// TwinCAT 3 PLC project P637_teljes
// ProgramVersion: 3.1.4023.0
// libraries:
//   Tc2_MC2, * (Beckhoff Automation GmbH)
//   Tc2_NC, * (Beckhoff Automation GmbH)
//   Tc2_SerialCom, * (Beckhoff Automation GmbH)
//   Tc2_Standard, * (Beckhoff Automation GmbH)
//   Tc2_System, * (Beckhoff Automation GmbH)
//   Tc2_TcpIp, * (Beckhoff Automation GmbH)
//   Tc2_Utilities, * (Beckhoff Automation GmbH)
//   Tc3_Module, * (Beckhoff Automation GmbH)
//   VisuDialogs, * (System)
//   Recipe Management,3.5.13.0,System
// project tree:
//   / CheckDivDInt.TcPOU, CheckDivLInt.TcPOU, CheckDivLReal.TcPOU, CheckDivReal.TcPOU, CheckLRangeSigned.TcPOU, CheckLRangeUnsigned.TcPOU, CheckPointer.TcPOU, CheckRangeSigned.TcPOU, CheckRangeUnsigned.TcPOU, GlobalTextList.TcGTLO, ImagePool.TcIPO (not stored), Jozsitengely_task.TcTTO, NTC_Task.TcTTO, Pistitengely_task.TcTTO, PlcTask.TcTTO, RecipeManager.TcRMO (not stored), Robot_task.TcTTO, Visualization Manager.TcVMO (not stored), VISU_TASK.TcTTO
//   DUTs/ ST_RobotState.TcDUT, STATES.TcDUT, User.TcDUT
//   GVLs/ GVL.TcGVL
//   POUs/ AUTOMATA.TcPOU, AUTOMATA_lepesek1.TcTLO, AUTOMATA_lepesek2.TcTLO, CheckBounds.TcPOU, DUT_types.TcTLO, ErrorList.TcTLO, ErrorList1.TcTLO, ErrorList2.TcTLO, JozsiProcess.TcPOU, MAIN.TcPOU
//   POUs/GENERAL/Components/ BARCODE_SCANNER.TcPOU, HEGESZTOK.TcPOU, INIT.TcPOU, RobotProcess.TcPOU, TERMEKVALTAS.TcPOU
//   POUs/GENERAL/Components/Robot/ ROBOTCOMMAND_OLD.TcPOU, ROBOTCOMMAND.TcPOU, ROBOTREMOTE_OLD.TcPOU, ROBOTREMOTE.TcPOU
//   POUs/GENERAL/Helpers/ fb_RobotStatusToBools.TcPOU, fb_SplitRobotResult.TcPOU, f_RobotCommandTranslation.TcPOU, f_RobotNTCTengelytolTavol.TcPOU, f_RobotPtTengelytolTavol.TcPOU, GetResourceFromCommand.TcPOU, f_GetRobotState.TcPOU
//   POUs/GENERAL/Executors/ f_E_Robot.TcPOU
//   POUs/JOZSI/Components/ HAJLITOK.TcPOU, HEGESZTESUTMERES.TcPOU, HEGESZTESUTMERES_1.TcPOU, HEGESZTOFEJTISZTITAS.TcPOU, JOZSITENGELY.TcPOU, KAMERA.TcPOU, NTC.TcPOU, NTCProcess.TcPOU
//   POUs/JOZSI/Executors/ f_E_Tengely.TcPOU
//   POUs/PISTI/Components/ KameraProcess.TcPOU, KAMERAREMOTE.TcPOU, KAPPE.TcPOU, HIMBA.TcPOU, Laser.TcPOU, Laser_old.TcPOU, LOGGING.TcPOU, PISTITENGELY.TcPOU, TEST_R_INTERPOL.TcPOU, ZEBRASCANNER.TcPOU, VEGMERO.TcPOU
//   POUs/PISTI/Helpers/ fb_GetPT1000MinMaxResFromTemp.TcPOU, f_GetNTCMinR.TcPOU, f_GetNTCMaxR.TcPOU, f_GetNTCNomR.TcPOU, f_GetPtMinR.TcPOU, f_GetPtMaxR.TcPOU, f_GetPtNomR.TcPOU, f_GetPtTfromR.TcPOU, f_GetPTTEMPFromRES.TcPOU, f_GetISOLvalue.TcPOU, f_GetNTCMaxTempFromRes.TcPOU, f_GetNTCNomTempFromRes.TcPOU, f_GetNTCMinTempFromRes.TcPOU, REAL_TO_STRING2.TcPOU
//   VISUs/ AddDelete.TcVIS, Biztos.TcVIS, Hegesztes_Karbantartas.TcVIS, Hegesztofej_IOk.TcVIS, Hegesztofej_IOk_Pt.TcVIS, Hegesztofej_IOk_NTC.TcVIS, Himba.TcVIS, Kamera_Pt.TcVIS, Login.TcVIS, Pt1000_oldali_kamera.TcVIS, Hegeszto_statusz.TcVIS, Lezer.TcVIS, Kamera.TcVIS, Robot.TcVIS, Kappe_pres.TcVIS, Start_ablak.TcVIS, Behelyezes.TcVIS, Rendszerinditas.TcVIS, Start_ellenorzes.TcVIS, Tengely_NTC_beallitasok.TcVIS, Tengely_Pt1000.TcVIS, Tengelyek.TcVIS, Tengely_NTC.TcVIS, Tengely_Pt1000_beallitasok.TcVIS, Termektipus.TcVIS, Vegmero.TcVIS, Hegesztes_Tengely_Pt1000.TcVIS, Hegesztes_Tengely_NTC.TcVIS, Kodolvaso.TcVIS, Hajlitok.TcVIS, Szerviz.TcVIS, NTC_szerviz.TcVIS, Hegesztok.TcVIS, Termeles0.TcVIS, Meresek.TcVIS, Beallitasok.TcVIS, Vegmero_idoallando.TcVIS, Vegmero_sokk.TcVIS, Vegmero_teljes.TcVIS, Vegmero_szigeteles.TcVIS, Vegmero_auto.TcVIS, Vegmero_ellenallas.TcVIS, Vegmero_kezi.TcVIS, Visualization_new.TcVIS
// real-time tasks:
//   TASK PlcTask: cycle T#10ms, priority 12, ADS port 350
//   TASK 637Visual: cycle T#20ms, priority 16, ADS port 351
//   TASK Pistitengely_task: cycle T#10ms, priority 13, ADS port 352
//   TASK Jozsitengely_task: cycle T#10ms, priority 14, ADS port 353
//   TASK Robot_task: cycle T#10ms, priority 20, ADS port 354
//   TASK NTC_Task: cycle T#1ms, priority 11, ADS port 355
//   TASK zebra: cycle T#1ms, priority 26, ADS port 356
// motion (NC):
//   TASK NC-Task 1 SAF: cycle T#2ms, priority 4, ADS port 501
//   TASK NC-Task 1 SVB: cycle T#2ms, priority 6, ADS port 511
//   AXIS JozsiTengely (id 1)
//     Dynamic: AccelerationMaximum=25000, DecelerationMaximum=25000, Acceleration=11382.8, Deceleration=11382.8, Jerk=114403
//     Velo: RefSearch=100, RefSync=5, SlowManual=57.2, FastManual=343.2, Fast=1144, Maximum=1144
//     OtherSettings: AllowMotionCmdToSlave=true, PulseDistancePos=200, PulseDistanceNeg=200
//     encoder EncType=19
//       EncPara: ScaleFactorNumerator=20, ScaleFactorDenominator=1048576, MaxCount=#xffffffff
//         Inc: RefMode=1
//     drive DrvType=16
//       DrvPara: MaxCount=#xffffffff, DriveControlDWord=#x00000100
//         Analog: VeloReferenz=1258.4
//         TimeComp: TaskDelayCycles=1
//     controller CtrType=1
//       CtrPara: PriorControlFactor=1
//         PosDiffControl: Enable=false, Range=200
//         Observer: BandWidth=20
//   AXIS PistiTengely (id 2)
//     Dynamic: Acceleration=11325.5840016781, Deceleration=11325.5840016781, Jerk=114411.676767905
//     Velo: RefSearch=100, RefSync=5, SlowManual=57.2, FastManual=343.2, Fast=1144, Maximum=1144
//     OtherSettings: AllowMotionCmdToSlave=true
//     encoder EncType=19
//       EncPara: ScaleFactorNumerator=20, ScaleFactorDenominator=1048576, MaxCount=#xffffffff
//         Inc: RefMode=1
//     drive DrvType=16
//       DrvPara: MaxCount=#xffffffff, DriveControlDWord=#x00000100
//         Analog: VeloReferenz=1200
//         TimeComp: TaskDelayCycles=1
//     controller CtrType=1
//       CtrPara: PriorControlFactor=1
//         PosDiffControl: Enable=false
//         Observer: BandWidth=20
// I/O:
//   DEVICE Device 1 (EtherCAT), AmsNetId 10.0.0.31.2.1
//     Term 1 (EK1200) [EK1200-5000 EtherCAT Power supply (2A E-Bus)]
//       PistiTengely (EL7211-0010) [EL7211-0010 1Ch. MDP742 Servo motor output stage with OCT (50V, 4.5A RMS)]
//       JózsiTengely (EL7211-0010) [EL7211-0010 1Ch. MDP742 Servo motor output stage with OCT (50V, 4.5A RMS)]
//       Útmérők 4 (EL5032) [EL5032 2Ch. EnDat Encoder]
//       Bemenetek (EL1809) [EL1809 16Ch. Dig. Input 24V, 3ms]
//       Bemenetek2 (EL1809) [EL1809 16Ch. Dig. Input 24V, 3ms]
//       Kimenetek (EL2809) [EL2809 16Ch. Dig. Output 24V, 0.5A]
//       Kimenetek2 (EL2809) [EL2809 16Ch. Dig. Output 24V, 0.5A]
//       Hőszenzor (EL3201-0010) [EL3201-0010 1K. Ana. Eingang PT100 (RTD), hochgenau]
//       EtherCatTerminal (EK1122) [EK1122 2 port EtherCAT junction]
//         Pisti Inputs1 (EP1008-0001) [EP1008-0001 8 Ch. Dig. Input 24V, 3ms, M8]
//         Pisti Inputs2 (EP1809-0021) [EP1809-0021 16 Ch. Dig. Input 24V, 3ms, M8]
//         IOLink Box (EP6224-3022) [EP6224-3022 (IO Link Master Class B)]
//         Jozsi Inputs1 (EP1809-0021) [EP1809-0021 16 Ch. Dig. Input 24V, 3ms, M8]
//         Jozsi Inputs2 (EP1809-0021) [EP1809-0021 16 Ch. Dig. Input 24V, 3ms, M8]
//         Végméro (EK1100) [EK1100 EtherCAT Coupler (2A E-Bus)]
//           AnalogIn (EL3068) [EL3068 8Ch. Ana. Input 0-10V]
//           DigitalIn (EL1808) [EL1808 8Ch. Dig. Input 24V, 3ms]
//           DigitalOut (EL2808) [EL2808 8Ch. Dig. Output 24V, 0.5A]
//           Term 18 (EL9011) [EL9011 End Terminal]
// variable links:
//   NC-Task 1 SAF/Axes/JozsiTengely <-> Device 1 (EtherCAT)/Term 1 (EK1200)/JózsiTengely (EL7211-0010)
//     Drive/Inputs/In/nDataIn1 <-> DRV Following error actual value/Following error actual value
//     Drive/Inputs/In/nDcOutputTime <-> InfoData/DcOutputShift
//     Drive/Inputs/In/nState1 <-> DRV Statusword/JozsiStatusword
//     Drive/Inputs/In/nState2 <-> DRV Statusword/JozsiStatusword @bit 8
//     Drive/Inputs/In/nState4 @bit 1 <-> WcState/InputToggle
//     Drive/Inputs/In/nState4 <-> WcState/WcState
//     Drive/Outputs/Out/nCtrl1 <-> DRV Controlword/Controlword
//     Drive/Outputs/Out/nCtrl2 <-> DRV Controlword/Controlword @bit 8
//     Drive/Outputs/Out/nDataOut1 <-> DRV Target position/Target position
//     Enc/Inputs/In/nDataIn1 <-> FB Position/Position
//     Enc/Inputs/In/nDcInputTime <-> InfoData/DcInputShift
//     Enc/Inputs/In/nState4 @bit 1 <-> WcState/InputToggle
//     Enc/Inputs/In/nState4 <-> WcState/WcState
//   NC-Task 1 SAF/Axes/PistiTengely <-> Device 1 (EtherCAT)/Term 1 (EK1200)/PistiTengely (EL7211-0010)
//     Drive/Inputs/In/nDataIn1 <-> DRV Following error actual value/Following error actual value
//     Drive/Inputs/In/nDcOutputTime <-> InfoData/DcOutputShift
//     Drive/Inputs/In/nState1 <-> DRV Statusword/PistiStatusword
//     Drive/Inputs/In/nState2 <-> DRV Statusword/PistiStatusword @bit 8
//     Drive/Inputs/In/nState4 @bit 1 <-> WcState/InputToggle
//     Drive/Inputs/In/nState4 <-> WcState/WcState
//     Drive/Outputs/Out/nCtrl1 <-> DRV Controlword/Controlword
//     Drive/Outputs/Out/nCtrl2 <-> DRV Controlword/Controlword @bit 8
//     Drive/Outputs/Out/nDataOut1 <-> DRV Target position/Target position
//     Enc/Inputs/In/nDataIn1 <-> FB Position/Position
//     Enc/Inputs/In/nDcInputTime <-> InfoData/DcInputShift
//     Enc/Inputs/In/nState4 @bit 1 <-> WcState/InputToggle
//     Enc/Inputs/In/nState4 <-> WcState/WcState
//   P637_teljes/P637_teljes Instance <-> Device 1 (EtherCAT)/Term 1 (EK1200)/Bemenetek (EL1809)
//     NTC_Task Inputs/GVL.bFenysorompoPt <-> Channel 15/FénysorompóPt
//     NTC_Task Inputs/HEGESZTOK.bHegesztoStromFehler <-> Channel 7/HegesztoStromFehler
//     NTC_Task Inputs/MAIN.bLevegoOK <-> Channel 3/LevegoOK
//     NTC_Task Inputs/NTC.bAlarm <-> Channel 12/NTC_Alarm
//     NTC_Task Inputs/NTC.bReady <-> Channel 13/NTC_Ready
//     PlcTask Inputs/GVL.bFenysorompoNTC <-> Channel 16/FénysorompóNTC
//     PlcTask Inputs/GVL.bHeatingTempOK <-> Channel 2/FűtőtőmbHőmOK
//     PlcTask Inputs/HEGESZTOK.bHegesztoBereit <-> Channel 6/HegesztoBereit
//     PlcTask Inputs/HEGESZTOK.bHegesztoFK <-> Channel 14/HegesztoFolyamatKesz
//     PlcTask Inputs/HEGESZTOK.bHegesztoMitStromIn <-> Channel 8/HegesztoMitStrom
//     PlcTask Inputs/VEGMERO.bFedelNyitva <-> Channel 1/VegmeroFedelLecsukásÉrzékelő
//     Robot_task Inputs/HEGESZTOK.bHegesztoElektrodenAnfordem <-> Channel 5/HegesztoElektrodenAnfordem
//     Robot_task Inputs/HEGESZTOK.bHegesztoNichtBereit <-> Channel 9/HegesztoNichtBereit
//     Robot_task Inputs/HEGESZTOK.bHegesztoVorwarnung <-> Channel 4/HegesztoVorwarnung
//     Robot_task Inputs/NTC.bSpeedReached <-> Channel 11/NTC_SpeedReached
//     Robot_task Inputs/NTC.bZeroSpeed <-> Channel 10/NTC_ZeroSpeed
//   P637_teljes/P637_teljes Instance <-> Device 1 (EtherCAT)/Term 1 (EK1200)/Bemenetek2 (EL1809)
//     PlcTask Inputs/GVL.bBiztonsagiFold <-> Channel 5/BiztonságiFöld
//     PlcTask Inputs/GVL.bBiztonsagiTap <-> Channel 6/BiztonságiTáp
//     PlcTask Inputs/GVL.bHegesztoHiba <-> Channel 7/HegesztoHiba
//     PlcTask Inputs/GVL.bKameraHulsePozOK <-> Channel 2/KameraHulsePoz
//     PlcTask Inputs/GVL.bKameraHulseVanOK <-> Channel 1/KameraHulseVan
//     PlcTask Inputs/GVL.bKameraSzinekOK <-> Channel 3/KameraSzinekOK
//     PlcTask Inputs/GVL.bKameraVezetekPozOK <-> Channel 4/KameraTavOK
//     PlcTask Inputs/HIMBA.bHimba_szenzor <-> Channel 10/Himba_szenzor
//     Robot_task Inputs/GVL.bPtKameraHegesztesOK <-> Channel 9/PtKameraHegesztesOK
//   P637_teljes/P637_teljes Instance <-> Device 1 (EtherCAT)/Term 1 (EK1200)/EtherCatTerminal (EK1122)/IOLink Box (EP6224-3022)
//     NTC_Task Outputs/HEGESZTOK.bHegeszto3 <-> IO-Link Port1/Hegeszto
//     NTC_Task Outputs/HEGESZTOK.bHegesztoFejekOutput[0] <-> IO-Link Port3/Hegesztofej1LE
//     NTC_Task Outputs/HEGESZTOK.bHegesztoFejekOutput[1] <-> IO-Link Port3/Hegesztofej2LE
//     NTC_Task Outputs/HEGESZTOK.bHegesztoFejekOutput[2] <-> IO-Link Port3/Hegesztofej3LE
//     NTC_Task Outputs/HEGESZTOK.bHegesztoFejekOutput[3] <-> IO-Link Port3/Valve 4 solenoid 14
//     PlcTask Outputs/GVL.bAdapterLefogo <-> IO-Link Port1/AdapterLefogó
//     PlcTask Outputs/HAJLITOK.bElohajlitoAlso <-> IO-Link Port4/AlsoElohajlito
//     PlcTask Outputs/HAJLITOK.bElohajlitoFelso <-> IO-Link Port4/FelsoElohajlito
//     PlcTask Outputs/HAJLITOK.bVeghajlitoAlso <-> IO-Link Port4/AlsoVeghajlito
//     PlcTask Outputs/HAJLITOK.bVeghajlitoFelso <-> IO-Link Port4/FelsoVeghajlito
//     PlcTask Outputs/HIMBA.bHimba <-> IO-Link Port1/Himba
//     PlcTask Outputs/KAPPE.bKappeBalFelLe <-> IO-Link Port1/KappeprésBal
//     PlcTask Outputs/KAPPE.bKappeFelLe <-> IO-Link Port1/Kappeprés
//     PlcTask Outputs/KAPPE.bKappeJobbFelLe <-> IO-Link Port1/KappeprésJobb
//     PlcTask Outputs/MAIN.bZoliSzelep <-> IO-Link Port4/Valve 5 solenoid 14
//     PlcTask Outputs/NTCProcess.bKiszedo <-> IO-Link Port2/NTC_Kiszedo
//     PlcTask Outputs/NTCProcess.bMegfogo <-> IO-Link Port2/NTC_Megfogo
//     PlcTask Outputs/NTCProcess.bVagoHajlito <-> IO-Link Port2/NTC_VagoHajlito
//     PlcTask Outputs/VEGMERO.bHutesOn <-> IO-Link Port1/HutesBe
//     PlcTask Outputs/VEGMERO.bLezertakaro <-> IO-Link Port1/LézerTakaró
//     PlcTask Outputs/VEGMERO.bMerotukBeKi <-> IO-Link Port1/Mérofej
//     PlcTask Outputs/VEGMERO.bPlatniBalraJobbra <-> IO-Link Port1/PlatniForgat
//     PlcTask Outputs/VEGMERO.bPlatniFelLe <-> IO-Link Port1/PlatniLeFel
//     Robot_task Outputs/GVL.bTempJozsiSzeleptombNTC[{3..7}] <-> IO-Link Port2/Valve {4..8} solenoid 14  (5 links)
//     Robot_task Outputs/GVL.bTempJozsiSzeleptomb[5] <-> IO-Link Port4/Valve 6 solenoid 14
//     Robot_task Outputs/GVL.bTempJozsiSzeleptomb[6] <-> IO-Link Port4/Valve 7 solenoid 14
//     Robot_task Outputs/GVL.bTempJozsiSzeleptomb[7] <-> IO-Link Port4/Valve 8 solenoid 14
//   P637_teljes/P637_teljes Instance <-> Device 1 (EtherCAT)/Term 1 (EK1200)/EtherCatTerminal (EK1122)/Jozsi Inputs1 (EP1809-0021)
//     Jozsitengely_task Inputs/GVL.bJozsiNegSwitch <-> Channel 7/LimitSwitchNeg
//     NTC_Task Inputs/NTC.bNTCLaberzekeloJobb <-> Channel 16/NTCJobbPozicioban
//     NTC_Task Inputs/NTC.bPirosGomb <-> Channel 13/NTCPirosGomb
//     NTC_Task Inputs/NTC.bZoldGomb <-> Channel 14/NTCZöldGomb
//     PlcTask Inputs/GVL.bHegeszto2FentBent <-> Channel 4/Hegeszto2FentBent
//     PlcTask Inputs/GVL.bHegeszto2FentKint <-> Channel 3/Hegeszto2FentKint
//     PlcTask Inputs/GVL.bHegeszto2LentBent <-> Channel 5/Hegeszto2LentBent
//     PlcTask Inputs/GVL.bHegeszto2LentKint <-> Channel 6/Hegeszto2LentKint
//     PlcTask Inputs/JOZSITENGELY.bNTC_OK <-> Channel 15/NTC_OK
//     PlcTask Inputs/NTCProcess.bKiszedoBent <-> Channel 12/NTC_KiszedoBent
//     PlcTask Inputs/NTCProcess.bKiszedoKint <-> Channel 11/NTC_KiszedoKint
//     PlcTask Inputs/NTCProcess.bMegfogoNyitva <-> Channel 9/NTC_MegfogoNyitva
//     PlcTask Inputs/NTCProcess.bMegfogoZarva <-> Channel 10/NTC_MegfogoZarva
//     PlcTask Inputs/NTCProcess.bVagoHajlitoFent <-> Channel 2/NTCVagoFent
//     PlcTask Inputs/NTCProcess.bVagoHajlitoLent <-> Channel 1/NTCVagoLent
//     Robot_task Inputs/GVL.bLimitSwitchNeg <-> Channel 7/LimitSwitchNeg
//     Robot_task Inputs/GVL.bNTCPirosGomb <-> Channel 13/NTCPirosGomb
//     Robot_task Inputs/GVL.bNTCPozicioban <-> Channel 8/NTCBalPozicioban
//     Robot_task Inputs/GVL.bNTCVagoFent <-> Channel 2/NTCVagoFent
//     Robot_task Inputs/GVL.bNTCVagoLent <-> Channel 1/NTCVagoLent
//     Robot_task Inputs/GVL.bNTCZoldGomb <-> Channel 14/NTCZöldGomb
//     Robot_task Inputs/GVL.bNTC_KiszedoBent <-> Channel 12/NTC_KiszedoBent
//     Robot_task Inputs/GVL.bNTC_KiszedoKint <-> Channel 11/NTC_KiszedoKint
//     Robot_task Inputs/GVL.bNTC_MegfogoNyitva <-> Channel 9/NTC_MegfogoNyitva
//     Robot_task Inputs/GVL.bNTC_MegfogoZarva <-> Channel 10/NTC_MegfogoZarva
//     Robot_task Inputs/GVL.bNTC_OK <-> Channel 15/NTC_OK
//     Robot_task Inputs/NTC.bNTCLaberzekeloBal <-> Channel 8/NTCBalPozicioban
//   P637_teljes/P637_teljes Instance <-> Device 1 (EtherCAT)/Term 1 (EK1200)/EtherCatTerminal (EK1122)/Jozsi Inputs2 (EP1809-0021)
//     Jozsitengely_task Inputs/GVL.bJozsiPosSwitch <-> Channel 16/LimitSwitchPlus
//     Jozsitengely_task Inputs/JOZSITENGELY.bJozsiHomeSwitch <-> Channel 16/LimitSwitchPlus
//     PlcTask Inputs/GVL.bHegeszto1BalFent <-> Channel 5/Hegeszto1BalFent
//     PlcTask Inputs/GVL.bHegeszto1BalLent <-> Channel 6/Hegeszto1BalLent
//     PlcTask Inputs/GVL.bHegeszto1JobbFent <-> Channel 13/Hegeszto1JobbFent
//     PlcTask Inputs/GVL.bHegeszto1JobbLent <-> Channel 14/Hegeszto1JobbLent
//     PlcTask Inputs/GVL.bNTCAdapterErzekelo <-> Channel 15/AdapterÉrzékelő
//     PlcTask Inputs/GVL.bPres1AlsoLent <-> Channel 3/Pres1AlsoLent
//     PlcTask Inputs/GVL.bPres2AlsoLent <-> Channel 12/Pres2AlsoLent
//     PlcTask Inputs/GVL.bPres1FelsoFent <-> Channel 2/Pres1FelsoFent
//     PlcTask Inputs/GVL.bPres2FelsoFent <-> Channel 10/Pres2FelsoFent
//     PlcTask Inputs/GVL.bStartNTC <-> Channel 8/StartNTC
//     PlcTask Inputs/HAJLITOK.bElohajlitoAlsoFent <-> Channel 4/Pres1AlsoFent
//     PlcTask Inputs/HAJLITOK.bElohajlitoAlsoLent <-> Channel 3/Pres1AlsoLent
//     PlcTask Inputs/HAJLITOK.bElohajlitoFelsoFent <-> Channel 2/Pres1FelsoFent
//     PlcTask Inputs/HAJLITOK.bElohajlitoFelsoLent <-> Channel 1/Pres1FelsoLent
//     PlcTask Inputs/HAJLITOK.bVeghajlitoAlsoFent <-> Channel 11/Pres2AlsoFent
//     PlcTask Inputs/HAJLITOK.bVeghajlitoAlsoLent <-> Channel 12/Pres2AlsoLent
//     PlcTask Inputs/HAJLITOK.bVeghajlitoFelsoFent <-> Channel 10/Pres2FelsoFent
//     PlcTask Inputs/HAJLITOK.bVeghajlitoFelsoLent <-> Channel 9/Pres2FelsoLent
//     PlcTask Inputs/MAIN.bZoliGomb <-> Channel 7/Input
//     Robot_task Inputs/GVL.bLimitSwitchPlus <-> Channel 16/LimitSwitchPlus
//     Robot_task Inputs/GVL.bPres1AlsoFent <-> Channel 4/Pres1AlsoFent
//     Robot_task Inputs/GVL.bPres2AlsoFent <-> Channel 11/Pres2AlsoFent
//     Robot_task Inputs/GVL.bPres1FelsoLent <-> Channel 1/Pres1FelsoLent
//     Robot_task Inputs/GVL.bPres2FelsoLent <-> Channel 9/Pres2FelsoLent
//   P637_teljes/P637_teljes Instance <-> Device 1 (EtherCAT)/Term 1 (EK1200)/EtherCatTerminal (EK1122)/Pisti Inputs1 (EP1008-0001)
//     NTC_Task Inputs/GVL.bHegeszto3Lent <-> Channel 5/HegesztőLent
//     Pistitengely_task Inputs/GVL.bPistiPosSwitch <-> Channel 6/LimitSwichPlus
//     Pistitengely_task Inputs/PISTITENGELY.bPistiHomeSwitch <-> Channel 6/LimitSwichPlus
//     PlcTask Inputs/GVL.bAdapterLefogoBent <-> Channel 1/AdapterLefogóBent
//     PlcTask Inputs/GVL.bAdapterLefogoKint <-> Channel 2/AdapterLefogóKint
//     PlcTask Inputs/GVL.bAdaptererzekelo <-> Channel 3/Adapterérzékelő
//     PlcTask Inputs/GVL.bHegeszto3Fent <-> Channel 4/HegesztőFent
//     PlcTask Inputs/HIMBA.bHimba_elol <-> Channel 8/Himba_elol
//     PlcTask Inputs/HIMBA.bHimba_hatul <-> Channel 7/Himba_hatul
//     Robot_task Inputs/GVL.bLimitSwichPlus <-> Channel 6/LimitSwichPlus
//     Robot_task Inputs/GVL.bTempPistiInputs1[0] <-> Channel 1/AdapterLefogóBent
//     Robot_task Inputs/GVL.bTempPistiInputs1[1] <-> Channel 2/AdapterLefogóKint
//     Robot_task Inputs/GVL.bTempPistiInputs1[2] <-> Channel 3/Adapterérzékelő
//     Robot_task Inputs/GVL.bTempPistiInputs1[3] <-> Channel 4/HegesztőFent
//     Robot_task Inputs/GVL.bTempPistiInputs1[4] <-> Channel 5/HegesztőLent
//     Robot_task Inputs/GVL.bTempPistiInputs1[5] <-> Channel 6/LimitSwichPlus
//   P637_teljes/P637_teljes Instance <-> Device 1 (EtherCAT)/Term 1 (EK1200)/EtherCatTerminal (EK1122)/Pisti Inputs2 (EP1809-0021)
//     Pistitengely_task Inputs/GVL.bPistiNegSwitch <-> Channel 8/LimitSwitchMinus
//     PlcTask Inputs/GVL.bKappePresFent <-> Channel 15/KappePrésFent
//     PlcTask Inputs/GVL.bKappepresNincsLegalul <-> Channel 7/KappeprésNincsLegalul
//     PlcTask Inputs/KAPPE.bKappeBalFent <-> Channel 11/KappeBalBent
//     PlcTask Inputs/KAPPE.bKappeBalLent <-> Channel 12/KappeBalKint
//     PlcTask Inputs/KAPPE.bKappeJobbFent <-> Channel 10/KappeJobbBent
//     PlcTask Inputs/KAPPE.bKappeJobbLent <-> Channel 9/KappeJobbKint
//     PlcTask Inputs/VEGMERO.bLezertakaroNyitva <-> Channel 6/LézerNyitva
//     PlcTask Inputs/VEGMERO.bLezertakaroZarva <-> Channel 5/LézerZárva
//     PlcTask Inputs/VEGMERO.bMerotukBent <-> Channel 4/MérőBent
//     PlcTask Inputs/VEGMERO.bMerotukKint <-> Channel 3/MérőKint
//     PlcTask Inputs/VEGMERO.bNagyFeszMerotuLent <-> Channel 16/NagyFeszMérőtűLent
//     PlcTask Inputs/VEGMERO.bPlatniBalon <-> Channel 14/PlatniBalon
//     PlcTask Inputs/VEGMERO.bPlatniFent <-> Channel 1/PlatniFent
//     PlcTask Inputs/VEGMERO.bPlatniJobbon <-> Channel 13/PlatniJobbon
//     PlcTask Inputs/VEGMERO.bPlatniLent <-> Channel 2/PlatniLent
//     Robot_task Inputs/GVL.bKappeBalBent <-> Channel 11/KappeBalBent
//     Robot_task Inputs/GVL.bKappeBalKint <-> Channel 12/KappeBalKint
//     Robot_task Inputs/GVL.bKappeJobbBent <-> Channel 10/KappeJobbBent
//     Robot_task Inputs/GVL.bKappeJobbKint <-> Channel 9/KappeJobbKint
//     Robot_task Inputs/GVL.bLezerNyitva <-> Channel 6/LézerNyitva
//     Robot_task Inputs/GVL.bLezerZarva <-> Channel 5/LézerZárva
//     Robot_task Inputs/GVL.bLimitSwitchMinus <-> Channel 8/LimitSwitchMinus
//     Robot_task Inputs/GVL.bMeroBent <-> Channel 4/MérőBent
//     Robot_task Inputs/GVL.bMeroKint <-> Channel 3/MérőKint
//     Robot_task Inputs/GVL.bPlatniBalon <-> Channel 14/PlatniBalon
//     Robot_task Inputs/GVL.bPlatniFent <-> Channel 1/PlatniFent
//     Robot_task Inputs/GVL.bPlatniJobbon <-> Channel 13/PlatniJobbon
//     Robot_task Inputs/GVL.bPlatniLent <-> Channel 2/PlatniLent
//     Robot_task Inputs/KAPPE.bKappeFent <-> Channel 15/KappePrésFent
//     Robot_task Inputs/KAPPE.bKappeNincsLegalul <-> Channel 7/KappeprésNincsLegalul
//   P637_teljes/P637_teljes Instance <-> Device 1 (EtherCAT)/Term 1 (EK1200)/EtherCatTerminal (EK1122)/Végméro (EK1100)/AnalogIn (EL3068)
//     PlcTask Inputs/VEGMERO.NTRES <-> AI Standard Channel 6/NTRES
//     PlcTask Inputs/VEGMERO.NTRES2 <-> AI Standard Channel 8/NTRES2
//     PlcTask Inputs/VEGMERO.PTRES <-> AI Standard Channel 5/PTRES
//     PlcTask Inputs/VEGMERO.U12V <-> AI Standard Channel 1/U12V
//     PlcTask Inputs/VEGMERO.U48V <-> AI Standard Channel 7/U48V
//     PlcTask Inputs/VEGMERO.U600V <-> AI Standard Channel 3/U600V
//     PlcTask Inputs/VEGMERO.U600VExt <-> AI Standard Channel 2/U600VEXT
//     PlcTask Inputs/VEGMERO.UISOL <-> AI Standard Channel 4/UISOL
//   P637_teljes/P637_teljes Instance <-> Device 1 (EtherCAT)/Term 1 (EK1200)/EtherCatTerminal (EK1122)/Végméro (EK1100)/DigitalOut (EL2808)
//     PlcTask Outputs/VEGMERO.PT_SOKK48V <-> Channel 3/PT-SOKK
//     PlcTask Outputs/VEGMERO.b600VBe <-> Channel 1/600VBe
//     PlcTask Outputs/VEGMERO.bRL_ISOL <-> Channel 2/RL-ISOL
//     Robot_task Outputs/GVL.bVentillatorok1Be <-> Channel 7/Ventillatorok1
//     Robot_task Outputs/GVL.bVentillatorok2Be <-> Channel 8/Ventillatorok2
//   P637_teljes/P637_teljes Instance <-> Device 1 (EtherCAT)/Term 1 (EK1200)/Hőszenzor (EL3201-0010)
//     PlcTask Inputs/VEGMERO.iHorzekelo <-> RTD/Value
//   P637_teljes/P637_teljes Instance <-> Device 1 (EtherCAT)/Term 1 (EK1200)/JózsiTengely (EL7211-0010)
//     Jozsitengely_task Inputs/JOZSITENGELY.nAxisStatus <-> DRV Statusword/JozsiStatusword
//   P637_teljes/P637_teljes Instance <-> Device 1 (EtherCAT)/Term 1 (EK1200)/Kimenetek (EL2809)
//     NTC_Task Outputs/HEGESZTOK.bHegesztoMitStromOut <-> Channel 15/HegesztoMitStrom
//     NTC_Task Outputs/HEGESZTOK.bHegesztoProgramValasztoOutput[0] <-> Channel 12/HegesztoPRG0
//     NTC_Task Outputs/HEGESZTOK.bHegesztoProgramValasztoOutput[1] <-> Channel 13/HegesztoPRG1
//     NTC_Task Outputs/HEGESZTOK.bHegesztoProgramValasztoOutput[2] <-> Channel 14/HegesztoPRG2
//     NTC_Task Outputs/HEGESZTOK.bHegesztoProgramValasztoOutput[3] <-> Channel 16/HegesztoPRG3
//     NTC_Task Outputs/HEGESZTOK.bHegesztoStart <-> Channel 10/HegesztoSTART
//     NTC_Task Outputs/HEGESZTOK.bHegesztoValtoOutput[0] <-> Channel 6/HegesztoValto1
//     NTC_Task Outputs/HEGESZTOK.bHegesztoValtoOutput[1] <-> Channel 7/HegesztoValto2
//     NTC_Task Outputs/HEGESZTOK.bHegesztoValtoOutput[2] <-> Channel 8/HegesztoValto3
//     PlcTask Outputs/GVL.bHegesztoHibaTorles <-> Channel 11/HegesztoMeldung
//     PlcTask Outputs/MAIN.bLevego <-> Channel 9/Levego
//     Robot_task Outputs/GVL.bTempOutputs[{0..4}] <-> Channel {1..5}/Output  (5 links)
//   P637_teljes/P637_teljes Instance <-> Device 1 (EtherCAT)/Term 1 (EK1200)/Kimenetek2 (EL2809)
//     NTC_Task Outputs/HEGESZTOK.bHegesztoProgramValasztoOutput[4] <-> Channel 8/HegesztoPRG4
//     NTC_Task Outputs/NTC.bForwardRotationStart <-> Channel 2/NTC_ForwardRotationStart
//     NTC_Task Outputs/NTC.bReverseRotationStart <-> Channel 3/NTC_ReverseRotationStart
//     NTC_Task Outputs/NTC.bServoON <-> Channel 1/NTC_ServoON
//     PlcTask Outputs/GVL.bBiztonsagiZarBe <-> Channel 7/BiztonságiZár
//     PlcTask Outputs/GVL.bElszivasBe <-> Channel 4/bElszivasBe
//     PlcTask Outputs/GVL.bKameraPROG <-> Channel 10/KameraPROG
//     PlcTask Outputs/GVL.bKameraTrigger <-> Channel 9/KameraTrigger
//     PlcTask Outputs/GVL.bPtKameraTrigger <-> Channel 13/PtKameraTrigger
//     Robot_task Outputs/NTC.bNTCFekBal <-> Channel 11/NTCLeftBreak
//     Robot_task Outputs/NTC.bNTCFekJobb <-> Channel 12/NTCRightBreak
//     Robot_task Outputs/NTC.bReset <-> Channel 6/NTC_Reset
//     Robot_task Outputs/NTC.bSpeed1 <-> Channel 5/NTC_Speed1
//   P637_teljes/P637_teljes Instance <-> Device 1 (EtherCAT)/Term 1 (EK1200)/PistiTengely (EL7211-0010)
//     Pistitengely_task Inputs/PISTITENGELY.nAxisStatus <-> DRV Statusword/PistiStatusword
//   P637_teljes/P637_teljes Instance <-> Device 1 (EtherCAT)/Term 1 (EK1200)/Útmérők 4 (EL5032)
//     NTC_Task Inputs/HEGESZTOK.ulHegeszto1Utmero <-> FB Inputs Channel 1/Hegeszto1 Position
//     NTC_Task Inputs/HEGESZTOK.ulHegeszto2Utmero <-> FB Inputs Channel 2/Hegeszto2 Position
//   P637_teljes/P637_teljes Instance <-> NC-Task 1 SAF/Axes/JozsiTengely
//     Jozsitengely_task Inputs/GVL.axisJozsiTengely.NcToPlc <-> Outputs/ToPlc
//     Jozsitengely_task Inputs/JOZSITENGELY.bOperational <-> Outputs/ToPlc/StateDWord/Operational
//     Jozsitengely_task Inputs/JOZSITENGELY.lrJozsiActPos <-> Outputs/ToPlc/ActPos
//     Jozsitengely_task Outputs/GVL.axisJozsiTengely.PlcToNc <-> Inputs/FromPlc
//     Robot_task Inputs/JOZSITENGELY.nJozsiErrorCode <-> Outputs/ToPlc/ErrorCode
//   P637_teljes/P637_teljes Instance <-> NC-Task 1 SAF/Axes/PistiTengely
//     Pistitengely_task Inputs/GVL.axisPistiTengely.NcToPlc <-> Outputs/ToPlc
//     Pistitengely_task Inputs/PISTITENGELY.bOperational <-> Outputs/ToPlc/StateDWord/Operational
//     Pistitengely_task Inputs/PISTITENGELY.lrPistiActPos <-> Outputs/ToPlc/ActPos
//     Pistitengely_task Outputs/GVL.axisPistiTengely.PlcToNc <-> Inputs/FromPlc
//     Robot_task Inputs/PISTITENGELY.nPistiErrorCode <-> Outputs/ToPlc/ErrorCode

CONFIGURATION P637_teljes
    RESOURCE PLC ON TwinCAT3
        TASK Jozsitengely_task(INTERVAL := T#10ms, PRIORITY := 14);
        TASK NTC_Task(INTERVAL := T#1ms, PRIORITY := 11);
        TASK Pistitengely_task(INTERVAL := T#10ms, PRIORITY := 13);
        TASK PlcTask(INTERVAL := T#10ms, PRIORITY := 12);
        TASK Robot_task(INTERVAL := T#10ms, PRIORITY := 20);
        TASK VISU_TASK(INTERVAL := T#20ms, PRIORITY := 16);
        PROGRAM JOZSITENGELY WITH Jozsitengely_task : JOZSITENGELY;
        PROGRAM NTC WITH NTC_Task : NTC;
        PROGRAM HEGESZTESUTMERES WITH NTC_Task : HEGESZTESUTMERES;
        PROGRAM ZEBRASCANNER WITH NTC_Task : ZEBRASCANNER;
        PROGRAM HEGESZTOK WITH NTC_Task : HEGESZTOK;
        PROGRAM PISTITENGELY WITH Pistitengely_task : PISTITENGELY;
        PROGRAM MAIN WITH PlcTask : MAIN;
        PROGRAM Laser WITH PlcTask : Laser;
        PROGRAM VEGMERO WITH PlcTask : VEGMERO;
        PROGRAM HAJLITOK WITH PlcTask : HAJLITOK;
        PROGRAM NTCProcess WITH PlcTask : NTCProcess;
        PROGRAM KAPPE WITH PlcTask : KAPPE;
        PROGRAM AUTOMATA WITH PlcTask : AUTOMATA;
        PROGRAM HEGESZTOFEJTISZTITAS WITH PlcTask : HEGESZTOFEJTISZTITAS;
        PROGRAM INIT WITH PlcTask : INIT;
        PROGRAM LOGGING WITH PlcTask : LOGGING;
        PROGRAM TERMEKVALTAS WITH PlcTask : TERMEKVALTAS;
        PROGRAM KAMERA WITH PlcTask : KAMERA;
        PROGRAM HIMBA WITH PlcTask : HIMBA;
        PROGRAM KameraProcess WITH PlcTask : KameraProcess;
        PROGRAM KAMERAREMOTE WITH PlcTask : KAMERAREMOTE;
        PROGRAM BARCODE_SCANNER WITH PlcTask : BARCODE_SCANNER;
        PROGRAM RobotProcess WITH Robot_task : RobotProcess;
        PROGRAM ROBOTREMOTE WITH Robot_task : ROBOTREMOTE;
        PROGRAM ROBOTCOMMAND WITH Robot_task : ROBOTCOMMAND;
        PROGRAM VisuElems_Visu_Prg WITH VISU_TASK : VisuElems.Visu_Prg;
    END_RESOURCE
END_CONFIGURATION

// ---- DUTs/ST_RobotState.TcDUT
TYPE ST_RobotState :
STRUCT
	sResult: STRING;
	bVakuumSzippantoFent: BOOL;
	bVakuumSzippantoLent: BOOL;
	bCsipeszNyitva: BOOL;
	bCsipeszZarva: BOOL;
	bVakuumA: BOOL;
	bVakuumB: BOOL;
	rX: REAL;
	rY: REAL;
	rZ: REAL;
	rU: REAL;
	sHand: STRING;
END_STRUCT
END_TYPE

// ---- DUTs/STATES.TcDUT
{attribute 'qualified_only'}
{attribute 'strict'}
TYPE STATES :
(
	enum_member := 0
);
END_TYPE

// ---- DUTs/User.TcDUT
TYPE User:
	STRUCT
		UserID: INT;
		UserNumber: STRING;
		UserName: STRING;
		UserLevel: INT;
		UserExist: BOOL;
	END_STRUCT
END_TYPE

// ---- GVLs/GVL.TcGVL
{attribute 'qualified_only'}
VAR_GLOBAL
	
	//Felhasználók beállítása
	AddDelButtonDis: BOOL;
	LogButtonsDis: BOOL;
	Logout_Button: BOOL;
	AddDeleteEnabled: BOOL;
	LoginEnabled: BOOL;
	
	UserID_Elozo: INT;
	UserID_Temp: INT;
	UserTemp: User;
	UserActual: User;
	UserNotFound: BOOL;
	UserModify: BOOL;
	UserDelete: BOOL;

	Biztos: BOOL;
	
	//Persistent data változói
	bStart_WrPer: BOOL;
	bError_WrPer: BOOL;
	fbWritePersistentData: WritePersistentData;
	bBusy_WrPer: BOOL;
	
	//System
	EngineExecuteList : ARRAY[1..5] OF STRING;
	bSettingsAutoSaveElozo: BOOL;
	bSettingsAutoSave: BOOL;
	
	//Temp
//	bTempInputs AT %I*: ARRAY [0..15] OF BOOL;
	bHeatingTempOK AT %I*: BOOL;
	bTempOutputs AT %Q*: ARRAY [0..15] OF BOOL;
	
	// Kamera I/O-k
	bKameraTrigger AT %Q*: BOOL;
	bKameraPROG AT %Q*: BOOL;
	bKameraBusy AT %I*: BOOL;
	bKameraHulseVanOK AT %I*: BOOL;
	bKameraHulsePozOK AT %I*: BOOL;
	bKameraSzinekOK AT %I*: BOOL;
	bKameraVezetekPozOK AT %I*: BOOL;
	bPtKameraTrigger AT %Q*: BOOL;
	bPtKameraHegesztesOK AT %I*: BOOL;
	
	// Hegesztő I/O-k
	bHegesztoHiba AT %I*: BOOL;
	bHegesztoHibaTorles AT %Q*: BOOL;

	// Hegesztési beállítás
	nWeldingDeformation1: DINT;
	nWeldingDeformation2: DINT;
	nWeldingDeformation3: DINT;
	nWeldingDeformation4: DINT;
	nWeldingDeformation5: DINT;
	bAutomaticWeldingStop1Elozo: BOOL;
	bAutomaticWeldingStop1: BOOL;
	bAutomaticWeldingStop2Elozo: BOOL;
	bAutomaticWeldingStop2: BOOL;
	bAutomaticWeldingStop3Elozo: BOOL;
	bAutomaticWeldingStop3: BOOL;
	bAutomaticWeldingStop4Elozo: BOOL;
	bAutomaticWeldingStop4: BOOL;
	bAutomaticWeldingStop5Elozo: BOOL;
	bAutomaticWeldingStop5: BOOL;
	nWeldingStopDistance1Elozo: DINT := 320;
	nWeldingStopDistance1: DINT := 320;
	nWeldingDistanceMin1Elozo: DINT := 320;
	nWeldingDistanceMin1: DINT := 320;
	nWeldingDistanceMax1Elozo: DINT := 320;
	nWeldingDistanceMax1: DINT := 320;
	nWeldingStopDistance2Elozo: DINT := 320;
	nWeldingStopDistance2: DINT := 320;
	nWeldingDistanceMin2Elozo: DINT := 320;
	nWeldingDistanceMin2: DINT := 320;
	nWeldingDistanceMax2Elozo: DINT := 320;
	nWeldingDistanceMax2: DINT := 320;
	nWeldingStopDistance3Elozo: DINT := 320;
	nWeldingStopDistance3: DINT := 320;
	nWeldingDistanceMin3Elozo: DINT := 320;
	nWeldingDistanceMin3: DINT := 320;
	nWeldingDistanceMax3Elozo: DINT := 320;
	nWeldingDistanceMax3: DINT := 320;
	nWeldingStopDistance4Elozo: DINT := 320;
	nWeldingStopDistance4: DINT := 320;
	nWeldingDistanceMin4Elozo: DINT := 320;
	nWeldingDistanceMin4: DINT := 320;
	nWeldingDistanceMax4Elozo: DINT := 320;
	nWeldingDistanceMax4: DINT := 320;
	nWeldingStopDistance5Elozo: DINT := 320;
	nWeldingStopDistance5: DINT := 320;
	nWeldingDistanceMin5Elozo: DINT := 320;
	nWeldingDistanceMin5: DINT := 320;
	nWeldingDistanceMax5Elozo: DINT := 320;
	nWeldingDistanceMax5: DINT := 320;
	nWeldingStopDistance1_637: DINT := 320;
	nWeldingDistanceMin1_637: DINT := 320;
	nWeldingDistanceMax1_637: DINT := 320;
	nWeldingStopDistance2_637: DINT := 320;
	nWeldingDistanceMin2_637: DINT := 320;
	nWeldingDistanceMax2_637: DINT := 320;
	nWeldingStopDistance3_637: DINT := 320;
	nWeldingDistanceMin3_637: DINT := 320;
	nWeldingDistanceMax3_637: DINT := 320;
	nWeldingStopDistance4_637: DINT := 320;
	nWeldingDistanceMin4_637: DINT := 320;
	nWeldingDistanceMax4_637: DINT := 320;
	nWeldingStopDistance5_637: DINT := 320;
	nWeldingDistanceMin5_637: DINT := 320;
	nWeldingDistanceMax5_637: DINT := 320;
	nWeldingStopDistance1_745: DINT := 320;
	nWeldingDistanceMin1_745: DINT := 320;
	nWeldingDistanceMax1_745: DINT := 320;
	nWeldingStopDistance2_745: DINT := 320;
	nWeldingDistanceMin2_745: DINT := 320;
	nWeldingDistanceMax2_745: DINT := 320;
	nWeldingStopDistance3_745: DINT := 320;
	nWeldingDistanceMin3_745: DINT := 320;
	nWeldingDistanceMax3_745: DINT := 320;
	nWeldingStopDistance4_745: DINT := 320;
	nWeldingDistanceMin4_745: DINT := 320;
	nWeldingDistanceMax4_745: DINT := 320;
	nWeldingStopDistance5_745: DINT := 320;
	nWeldingDistanceMin5_745: DINT := 320;
	nWeldingDistanceMax5_745: DINT := 320;
	ulWeldingStartDistance1: ULINT;
	ulWeldingStartDistance2: ULINT;
	ulWeldingStartDistance3: ULINT;
	ulWeldingStartDistance4: ULINT;
	ulWeldingStartDistance5: ULINT;
	nWeldingDistanceStartMin1Elozo: DINT := 0;
	nWeldingDistanceStartMin1: DINT := 0;
	nWeldingDistanceStartMax1Elozo: DINT := 210000;
	nWeldingDistanceStartMax1: DINT := 210000;
	nWeldingDistanceStartMin2Elozo: DINT := 0;
	nWeldingDistanceStartMin2: DINT := 0;
	nWeldingDistanceStartMax2Elozo: DINT := 210000;
	nWeldingDistanceStartMax2: DINT := 210000;
	nWeldingDistanceStartMin3Elozo: DINT := 0;
	nWeldingDistanceStartMin3: DINT := 0;
	nWeldingDistanceStartMax3Elozo: DINT := 210000;
	nWeldingDistanceStartMax3: DINT := 210000;
	nWeldingDistanceStartMin4Elozo: DINT := 0;
	nWeldingDistanceStartMin4: DINT := 0;
	nWeldingDistanceStartMax4Elozo: DINT := 210000;
	nWeldingDistanceStartMax4: DINT := 210000;
	nWeldingDistanceStartMin5Elozo: DINT := 0;
	nWeldingDistanceStartMin5: DINT := 0;
	nWeldingDistanceStartMax5Elozo: DINT := 210000;
	nWeldingDistanceStartMax5: DINT := 210000;
	bWeldingLog: BOOL;
	bWeldingLogElozo: BOOL;
	nElectrode1UsageElozo: DINT;
	nElectrode1Usage: DINT;
	nElectrode1UsageMaxElozo: DINT := 1;
	nElectrode1UsageMax: DINT := 1;
	nElectrode1UsageWarnElozo: DINT := 1;
	nElectrode1UsageWarn: DINT := 1;
	nElectrode1AlarmColor: DWORD := 16#FFFFFF00;
	nElectrode2UsageElozo: DINT;
	nElectrode2Usage: DINT;
	nElectrode2UsageMaxElozo: DINT := 1;
	nElectrode2UsageMax: DINT := 1;
	nElectrode2UsageWarnElozo: DINT := 1;
	nElectrode2UsageWarn: DINT := 1;
	nElectrode2AlarmColor: DWORD := 16#FF8F8F00;
	nElectrode3UsageElozo: DINT;
	nElectrode3Usage: DINT;
	nElectrode3UsageMaxElozo: DINT := 1;
	nElectrode3UsageMax: DINT := 1;
	nElectrode3UsageWarnElozo: DINT := 1;
	nElectrode3UsageWarn: DINT := 1;
	nElectrode3AlarmColor: DWORD := 16#FF8F8F00;
	
	nHegFejTisztCiklusokElozo: UINT := 5;
	nHegFejTisztCiklusok: UINT := 5;
	nHegFejTisztProgramElozo: UINT := 11;
	nHegFejTisztProgram: UINT := 11;
	
	//Pisti Globals
	axisPistiTengely: AXIS_REF;
	bPistiPosSwitch AT %I*: BOOL;
	bPistiNegSwitch AT %I*: BOOL;
	bPistiServo : BOOL := TRUE;
	bTempPistiInputs1 AT %I*: ARRAY [0..7] OF BOOL;
	bHimbaOK: BOOL := FALSE;
	bAdapterLefogoBent AT %I*: BOOL; // 0
	bAdapterLefogoKint AT %I*: BOOL; // 1
	bAdaptererzekelo AT %I*: BOOL; // 2
	bHegeszto3Fent AT %I*: BOOL; // 3
	bHegeszto3Lent AT %I*: BOOL; // 4
	bLimitSwichPlus AT %I*: BOOL; // 5
	bStartPt AT %I*: BOOL; // 6
	bInput_7: BOOL; // 7 
//	bTempPistiInputs2 AT %I*: ARRAY [0..15] OF BOOL;
	bPlatniFent AT %I*: BOOL; // 0
	bPlatniLent AT %I*: BOOL; // 1
	bMeroKint AT %I*: BOOL; // 2
	bMeroBent AT %I*: BOOL; // 3
	bLezerZarva AT %I*: BOOL; // 4
	bLezerNyitva AT %I*: BOOL; // 5
	bKappepresNincsLegalul AT %I*: BOOL; // 6
	bLimitSwitchMinus AT %I*: BOOL; // 7
	bKappeJobbKint AT %I*: BOOL; // 8
	bKappeJobbBent AT %I*: BOOL; // 9
	bKappeBalBent AT %I*: BOOL; // 10
	bKappeBalKint AT %I*: BOOL; // 11
	bPlatniJobbon AT %I*: BOOL; // 12
	bPlatniBalon AT %I*: BOOL; // 13
	bKappePresFent AT %I*: BOOL; // 14
	bInput_15: BOOL; // 15
//	bTempPistiOutputs1 AT %Q*: ARRAY [0..9] OF BOOL;
	bAdapterLefogo AT %Q*: BOOL; // 0
	bJOZSITENGELYReserved: BOOL;
	lrPtSzervizboxElozo : LREAL := -5;
	lrPtSzervizbox : LREAL := -5;
	lrNTCSzervizboxElozo : LREAL := -10;
	lrNTCSzervizbox : LREAL := -10;
	lrHajlitoPosition1Elozo : LREAL := -401.2;
	lrHajlitoPosition1 : LREAL := -401.2;
	lrHajlitoPosition2Elozo : LREAL := -575.1;
	lrHajlitoPosition2 : LREAL := -575.1;
	lrHegesztoPosition1Elozo : LREAL := -789.0;
	lrHegesztoPosition1 : LREAL := -789.0;
	lrHegesztoPosition2Elozo : LREAL := -792.0;
	lrHegesztoPosition2 : LREAL := -792.0;
	lrHegesztoPosition3Elozo : LREAL := -794.7;
	lrHegesztoPosition3 : LREAL := -794.7;
	lrCsiszoloPosition1Elozo : LREAL := -780;
	lrCsiszoloPosition1 : LREAL := -780;
	lrCsiszoloPosition2Elozo : LREAL := -800;
	lrCsiszoloPosition2 : LREAL := -800;
	lrHegesztoPosition4Elozo : LREAL := -1109.913;
	lrHegesztoPosition4 : LREAL := -1109.913;
	lrHegesztoPosition5Elozo : LREAL := -1101.15;
	lrHegesztoPosition5 : LREAL := -1101.15;
	lrHegesztoPosition6Elozo : LREAL := -379.7;
	lrHegesztoPosition6 : LREAL := -379.7;
	lrHegesztoPosition7Elozo : LREAL := -386;
	lrHegesztoPosition7 : LREAL := -386;
	lrNTCKameraPositionElozo : LREAL := -160.622;
	lrNTCKameraPosition : LREAL := -160.622;
	lrPtKameraPositionElozo : LREAL := -503.4;
	lrPtKameraPosition : LREAL := -503.4;
	lrRobotKappePositionElozo : LREAL := -694.5;
	lrRobotKappePosition : LREAL := --694.5;
	lrKodolvasasPositionElozo: LREAL := -841.54;
	lrKodolvasasPosition: LREAL := -841.54;
	lrKodolvasasPosition2Elozo: LREAL := -841.54;
	lrKodolvasasPosition2: LREAL := -841.54;
	lrKappePositionElozo : LREAL := -837.11;
	lrKappePosition : LREAL := -837.11;
	lrVegmeroPositionElozo : LREAL := -1054.776;
	lrVegmeroPosition : LREAL := -1054.776;
	
	//Jozsi Globals
	axisJozsiTengely: AXIS_REF;
	bJozsiPosSwitch AT %I*: BOOL;
	bJozsiNegSwitch AT %I*: BOOL;
	bJozsiServo : BOOL := TRUE;
//	bTempJozsiInputs1 AT %I*: ARRAY [0..15] OF BOOL;
	bNTCVagoLent AT %I*: BOOL; // 0
	bNTCVagoFent AT %I*: BOOL; // 1
	bHegeszto2FentKint AT %I*: BOOL; // 2
	bHegeszto2FentBent AT %I*: BOOL; // 3
	bHegeszto2LentBent AT %I*: BOOL; // 4
	bHegeszto2LentKint AT %I*: BOOL; // 5
	bLimitSwitchNeg AT %I*: BOOL; // 6
	bNTCPozicioban AT %I*: BOOL; // 7
	bNTC_MegfogoNyitva AT %I*: BOOL; // 8
	bNTC_MegfogoZarva AT %I*: BOOL; // 9
	bNTC_KiszedoKint AT %I*: BOOL; // 10
	bNTC_KiszedoBent AT %I*: BOOL; // 11
	bNTCPirosGomb AT %I*: BOOL; // 12
	bNTCZoldGomb AT %I*: BOOL; // 13
	bNTC_OK AT %I*: BOOL; // 14
	bNC_15: BOOL; // 15
//	bTempJozsiInputs2 AT %I*: ARRAY [0..15] OF BOOL;
	bPres1FelsoLent AT %I*: BOOL; // 0
	bPres1FelsoFent AT %I*: BOOL; // 1
	bPres1AlsoLent AT %I*: BOOL; // 2
	bPres1AlsoFent AT %I*: BOOL; // 3
	bHegeszto1BalFent AT %I*: BOOL; // 4
	bHegeszto1BalLent AT %I*: BOOL; // 5
	bStartNTC AT %I*: BOOL; // 6
	bInput7: BOOL; // 7
	bPres2FelsoLent AT %I*: BOOL; // 8
	bPres2FelsoFent AT %I*: BOOL; // 9
	bPres2AlsoFent AT %I*: BOOL; // 10
	bPres2AlsoLent AT %I*: BOOL; // 11
	bHegeszto1JobbFent AT %I*: BOOL; // 12
	bHegeszto1JobbLent AT %I*: BOOL; // 13
	bNTCAdapterErzekelo AT %I*: BOOL; // 14
	bLimitSwitchPlus AT %I*: BOOL; // 15
	bTempJozsiSzeleptombNTC AT %Q*: ARRAY [0..7] OF BOOL;
	bTempJozsiSzeleptomb AT %Q*: ARRAY [0..7] OF BOOL;
	bPISTITENGELYReserved: BOOL;
	bHegesztofejTisztitas: BOOL := FALSE;
	
	
	
	//Laser
	bLaserCommOpen : BOOL := FALSE;
	
	//Recipe Manager
	RecipeManagerCommands: RecipeManCommands;
	
	//Mérés
	bEtalonOn : BOOL := TRUE;
	bFedelOK : BOOL :=FALSE;
	bPTResOK : BOOL := FALSE;
	iPTResQ : BYTE :=0;
	bNTCResOK : BOOL := FALSE;
	bNTCRes2OK : BOOL := FALSE;
	iNTCResQ : BYTE := 0;
	iNTC2ResQ : BYTE := 0;
	bIsolOK : BOOL := FALSE;
	iIsolQ : BYTE := 0;
	bTimeConstOK : BOOL := FALSE;
	iTimeConstQ : BYTE := 0;
	bShockOK : BOOL := FALSE;
	iShockQ : BYTE := 0;
	bMarkingOK : BOOL := FALSE;
	bMarking_ellenorizve : BOOL;
	iMarkingQ : BYTE := 0;
	bProduct1OK : BOOL := FALSE;
	bProduct1NOK : BOOL := FALSE;
	bProductOK : BOOL := FALSE;
	bProductNOK : BOOL := FALSE;
	rTemp : REAL := 0;
	rPtRes : REAL := 0;
	rPtResShock : REAL;
	rPtDevElozo : REAL := 2;
	rPtDev : REAL := 2;
	rNTCRes : REAL :=0;
	rNTCRes2 : REAL :=0;
	rNTCDevElozo : REAL := 7;
	rNTCDev : REAL := 7;
	rNTC2DevElozo : REAL := 7;
	rNTC2Dev : REAL := 7;
	rISOL_MAXElozo : REAL := 0.97;
	rISOL_MAX : REAL := 0.97;
	rTempMaxElozo : REAL := 300.0;	// Fűtőtömb hőmérséklete
	rTempMax : REAL := 300.0;	// Fűtőtömb hőmérséklete
	rIdoallandoMaxElozo : REAL :=6;
	rIdoallandoMax : REAL :=6;
	rTimeConst : REAL :=0;
	PTRES_SOKK_MAXElozo : REAL := 2000.0;
	PTRES_SOKK_MAX : REAL := 2000.0;
	iSelectedProductType: INT :=-1;
	iPreviousSelectedProductType: INT :=-1;
	iCurrentProductType: INT :=-3;
	
	//Termelés
	nProductCount1 : DINT;
	nGoodProductCount1 : DINT;
	nBadProductCount1 : DINT;
	nGoodProductCount : DINT;
	nBadProductCount : DINT;
	sProductTypeName : STRING;
	saProductTypeNames: ARRAY[-3..0] OF STRING := ['6379XX_ETALON1', '6379XX_ETALON2',
					 '6379XX_ETALON3','637900'];
	saProductTypeNames745: ARRAY[-3..0] OF STRING := ['7459XX_ETALON1', '7459XX_ETALON2',
					 '7459XX_ETALON3','745900'];
	sNTCType: STRING;
	sPtType: STRING;
	sProductType: STRING;
	sNTCTypeElozo: STRING;
	sPtTypeElozo: STRING;
	sProductTypeElozo: STRING;
	bProductTypeOK: BOOL;

	bElszivasBe AT %Q*: BOOL;
	bSystemStarted: BOOL := FALSE;
	bSystemNotStarted: BOOL := TRUE;

	bHimbaBe: BOOL := FALSE;
	bKameraBe: BOOL := TRUE;
	bHajlitasBe: BOOL := TRUE;
	bHegesztes1Be: BOOL := TRUE;
	bHegesztes2Be: BOOL := TRUE;
	bHegesztes3Be: BOOL := TRUE;
	bHegesztes4Be: BOOL := TRUE;
	bHegesztes5Be: BOOL := TRUE;
	bKameraVegBe: BOOL := TRUE;
	bHegesztes6Be: BOOL := TRUE;
	bHegesztes7Be: BOOL := TRUE;
	bPtKameraBe: BOOL := FALSE;
	bRobotKappeBe: BOOL := TRUE;
	bKappeBe: BOOL := TRUE;
	bMeresBe: BOOL := TRUE;
	bJelolesBe: BOOL := TRUE;
	bNTCInditasFenysorompoval: BOOL;
	bPtInditasFenysorompoval: BOOL;
	sNTCKameraImageID: STRING := 'NTCKamera_NG_Image';
	iBitmap_Version: INT :=0;
	bNTCKameraElfogadva: BOOL := FALSE;
	bNTCKameraNemJo: BOOL := FALSE;
	bNTCEredmenyGombokRejtve: BOOL := TRUE;
	bNTCBezarGombRejtve: BOOL := TRUE;

	// Dátum, időpont
	sYear: STRING;
	sMonth: STRING;
	sDay: STRING;
	sHour: STRING;
	sMinute: STRING;
	sSecond: STRING;
	sDateTime: STRING;
	
	// GUI kezelés
	bMeresiEredmenyekRejtve: BOOL := TRUE;
	bKameraEredmenyekRejtve: BOOL := TRUE;
	bRegiFelulet: BOOL := FALSE;
	iFoLapozo: INT;
	iSzervizLapozo: INT;
	iTengelyLapozo: INT;
	iHegesztoLapozo: INT;
	iMeresLapozo: INT;
	iAutoMeresLapozo: INT;
	
	// Hibakezelés
	bHibauzenetNTCRejtve: BOOL;
	bHibauzenetPtRejtve: BOOL;
	bHibauzenetKozosRejtve: BOOL;
	nHibaKodNTC: UINT;
	nHibaKodPt: UINT;
	nHibaKodKozos: UINT;
	
	// Robot állapot
	stRobotStatusz: ST_RobotState;
	bRobotPaused: BOOL;
	
	// Biztonság
	bFenysorompoNTC AT %I*: BOOL;
	bFenysorompoPt AT %I*: BOOL;
	bBiztonsagiFold AT %I*: BOOL;
	bBiztonsagiTap AT %I*: BOOL;
	bBiztonsagiZarBe AT %Q*: BOOL;
	bVentillatorok1Be AT %Q*: BOOL := TRUE;
	bVentillatorok2Be AT %Q*: BOOL := TRUE;
	
	bBiztonsagiZarGomb: BOOL;
	nHibaKodRobot: UINT;
END_VAR
VAR_GLOBAL CONSTANT
	saProductTypes: ARRAY[-1..16] OF STRING := ['', '637900', '637910', '637920', '637930', '637901', '637911', '637921', '637931','521950','745900','745910','745905','745915','745906','745916','745907','745917'];
	NTC_Sensing_NomRT: ARRAY[0..1, 0..25] OF REAL := 
	[15, 16, 17, 18, 19, 20, 21, 22, 23, 24, 25, 26, 27, 28, 29, 30, 31, 32, 33, 34, 35, 36, 37, 38, 39, 40,
	15660.6, 14955.5, 14286.1, 13650.4, 13046.5, 12472.7, 11927.3, 11408.7, 10915.6, 10446.4, 10000, 9575.1, 9170.5, 8785.3, 8418.3, 8068.6, 7735.3, 7417.5, 7114.5, 6825.5, 6549.8, 6286.7, 6035.5, 5795.6, 5566.6, 5347.8];
	Pt_NomRT: ARRAY[0..1, 0..15] OF REAL := 
	[0,20,40,60,80,100,120,140,160,180,200,220,240,260,280,300,
	1000,1077.9,1155.4,1232.4,1309,1385.1,1460.7,1535.8,1610.5,1684.8,1758.6,1831.9,1904.7,1977.1,2049.1,2120.5];
	
	TERMELES_FUL: INT := 0;
	BEALLITASOK_FUL: INT := 1;
	SZERVIZ_FUL: INT := 2;
	RENDSZERIND_FUL: INT :=0;
	BEHELYEZES_FUL: INT := 1;
	TENGELYEK_FUL: INT := 2;
		NTC_TENGELY_FUL: INT := 0;
		PT_TENGELY_FUL: INT := 1;
	HAJLITOK_FUL: INT := 3;
	HEGESZTES_FUL: INT := 4;
		HEGESZTO_STATUSZ_FUL: INT := 2;
	ROBOT_FUL: INT := 5;
	NTC_VAGO_FUL: INT := 6;
	KAPPE_PRES_FUL: INT := 7;
	VEGMERO_FUL: INT := 8;
	LEZER_FUL: INT := 9;
	KODOLVASO_FUL: INT := 10;
	
	UserLevels: ARRAY[0..3] OF STRING := ['N/A', 'Operátor', 'Csoportvezető', 'Admin'];
	
END_VAR
VAR_GLOBAL PERSISTENT
	Users: ARRAY[0..99] OF User;
END_VAR

// ---- POUs/JOZSI/Components/JOZSITENGELY.TcPOU
PROGRAM JOZSITENGELY
VAR
	JozsiHome: MC_Home;
	bJozsiHomeEnable: BOOL := FALSE;
	bAxisBusy : BOOL := FALSE;
	bAxisActive: BOOL := FALSE;
	bAxisAborted: BOOL := FALSE;
	bAxisError: BOOL := FALSE;
	nAxisErrorID: UDINT;
	bAxisStopDone: BOOL := FALSE;
	bJozsiHomeSwitch AT %I*: BOOL;
	fbJozsiTengelyStop: MC_Stop;
	fbJozsitengelyServo: MC_Power;
	bJozsiPosSwitch : BOOL := TRUE;
	bJozsiTengelySzabad : BOOL;
	bOperational AT %I*: BOOL;
	bNTC_OK AT %I*: BOOL;
	bHomeReady : BOOL := FALSE;
	nAxisStatus AT %I*: UINT;
	bAxisReady : BOOL;
	bAxisOn : BOOL;
	
	//HOME
	bAxisHomeDone: BOOL;
	bAxisHomeBusy: BOOL;
	bAxisHomeActive: BOOL;
	bAxisHomeAborted: BOOL;
	bAxisHomeError: BOOL;
	nAxisHomeErrorID: UDINT;
	
	//MOVE
	bAxisMoveDone: BOOL;
	bAxisMoveBusy: BOOL;
	bAxisMoveActive: BOOL;
	bAxisMoveAborted: BOOL;
	bAxisMoveError: BOOL;
	nAxisMoveErrorID: UDINT;
	
	//COMMAND
	bAxisCommandDone: BOOL;
	bAxisCommandBusy: BOOL;
	bAxisCommandActive: BOOL;
	bAxisCommandAborted: BOOL;
	bAxisCommandError: BOOL;
	nAxisCommandErrorID: UDINT;
	
	
	fbJozsitengelyJOG: MC_Jog;
	bJozsiJOGPlus : BOOL := FALSE;
	bJozsiJOGMinus : BOOL := FALSE;
	fbJozsitengelyReset: MC_Reset;
	bJozsiReset: BOOL;
	nJozsiErrorCode AT %I*: UDINT;
	lrJozsiActPos AT %I*: LREAL;
	fbJozsiMoveAbsolute: MC_MoveAbsolute;
	
	//Pozíciók
//	lrSzervizbox : LREAL := -10;
//	lrHajlitoPosition1 : LREAL := -401.510;
//	lrHajlitoPosition2 : LREAL := -575.44;
//	lrHegesztoPosition1 : LREAL := -789.1;
//	lrHegesztoPosition2 : LREAL := -792.3;
//	lrHegesztoPosition3 : LREAL := -795.1;
//	lrHegesztoPosition4 : LREAL := -1109.913;
//	lrHegesztoPosition5 : LREAL := -1101.15;
//	lrSardisajatPosition1 : LREAL := -756;
//	lrSardisajatPosition2 : LREAL := -738;
	lrSardisajatPosition1 : LREAL := -656;
	lrSardisajatPosition2 : LREAL := -638;
	bJozsiTengelySzabad_TON: TON;
END_VAR
VAR_INPUT
	lrJozsiPosition : LREAL := 0;
	sJozsiAxisCommand: STRING := '';	
END_VAR
VAR_OUTPUT
	n_OutErrId: UINT;
END_VAR

bJozsiTengelySzabad := GVL.bPres1AlsoLent AND GVL.bPres1FelsoFent
						AND GVL.bPres2FelsoFent AND GVL.bPres2AlsoLent
						AND ((GVL.bHegeszto1BalFent AND GVL.bHegeszto1JobbFent) OR GVL.bHegesztofejTisztitas)
						AND GVL.bHegeszto2FentBent AND GVL.bHegeszto2LentBent AND bOperational
//						AND ((GVL.stRobotStatusz.rX>-100) 
//								OR (GVL.stRobotStatusz.rY>350)
//								OR (GVL.stRobotStatusz.rZ>-111))
						AND f_RobotNTCTengelytolTavol()
						AND (GVL.bFenysorompoNTC
							OR (sJozsiAxisCommand='HOME')
							OR (JOZSITENGELY.lrJozsiActPos>-10)
							OR (JOZSITENGELY.lrJozsiActPos<-500))
						AND NOT GVL.bBiztonsagiFold AND GVL.bBiztonsagiTap;
bJozsiTengelySzabad_TON(IN:=bJozsiTengelySzabad, PT:=T#100MS);
IF bJozsiTengelySzabad_TON.Q = FALSE THEN
	IF MAIN.bLevegoOK=FALSE THEN
		n_OutErrId := 5;
	ELSIF GVL.bPres1AlsoLent=FALSE THEN
		n_OutErrId := 149;
	ELSIF GVL.bPres1FelsoFent=FALSE THEN
		n_OutErrId := 147;
	ELSIF GVL.bPres2FelsoFent=FALSE THEN
		n_OutErrId := 163;
	ELSIF GVL.bPres2AlsoLent=FALSE THEN
		n_OutErrId := 167;
	ELSIF GVL.bHegeszto1BalFent=FALSE THEN
		n_OutErrId := 153;
	ELSIF GVL.bHegeszto1JobbFent=FALSE THEN
		n_OutErrId := 169;
	ELSIF GVL.bHegeszto2FentBent=FALSE THEN
		n_OutErrId := 119;
	ELSIF GVL.bHegeszto2LentBent=FALSE THEN
		n_OutErrId := 121;
	ELSIF bOperational=FALSE THEN
		n_OutErrId := 193;
//	ELSIF NOT ((GVL.stRobotStatusz.rX>-100)
//		OR (GVL.stRobotStatusz.rY>350)
//		OR (GVL.stRobotStatusz.rZ>-111)) THEN
	ELSIF NOT f_RobotNTCTengelytolTavol() THEN
		n_OutErrId := 302;
	ELSIF GVL.bFenysorompoNTC=FALSE THEN
		n_OutErrId := 31;
	ELSIF GVL.bBiztonsagiFold=TRUE THEN
		n_OutErrId := 42;
	ELSIF GVL.bBiztonsagiTap=FALSE THEN
		n_OutErrId := 43;
	END_IF
ELSE
	n_OutErrId := 0;
END_IF
bAxisReady:=nAxisStatus MOD 2 = 1;
bAxisOn:=nAxisStatus/2 MOD 2 = 1;

fbJozsiTengelyStop(
	Axis:= GVL.axisJozsiTengely, 
	Execute:= (NOT((GVL.bJozsiPosSwitch OR sJozsiAxisCommand='HOME') AND GVL.bJozsiNegSwitch AND bJozsiTengelySzabad_TON.Q)
				OR (sJozsiAxisCommand='STOP')), 
	Deceleration:= , 
	Jerk:= , 
	Options:= , 
	Done=> bAxisStopDone, 
	Busy=> bAxisBusy, 
	Active=> bAxisActive, 
	CommandAborted=> bAxisAborted, 
	Error=> bAxisError, 
	ErrorID=> nAxisErrorID);
IF (sJozsiAxisCommand='STOP') AND bAxisStopDone AND NOT bAxisError THEN
	sJozsiAxisCommand := '';
END_IF
IF NOT(GVL.bJozsiPosSwitch OR sJozsiAxisCommand='HOME') OR NOT(GVL.bJozsiNegSwitch) THEN
	GVL.bJozsiServo := FALSE;
	sJozsiAxisCommand:='';
END_IF
fbJozsitengelyServo(
	Axis:= GVL.axisJozsiTengely, 
	Enable:= GVL.bJozsiServo, 
	Enable_Positive:= (GVL.bJozsiPosSwitch OR sJozsiAxisCommand='HOME'), 
	Enable_Negative:= GVL.bJozsiNegSwitch, 
	Override:= 100, 
	BufferMode:= , 
	Options:= , 
	Status=> , 
	Busy=> , 
	Active=> , 
	Error=> , 
	ErrorID=> );
	
	//Home
JozsiHome(
	Axis:= GVL.axisJozsiTengely, 
	Execute:= sJozsiAxisCommand='HOME' AND bJozsiTengelySzabad_TON.Q, 
	Position:= DEFAULT_HOME_POSITION, 
	HomingMode:= MC_DefaultHoming, 
	BufferMode:= , 
	Options:= , 
	bCalibrationCam:= NOT(bJozsiHomeSwitch), 
	Done=> bAxisHomeDone, 
	Busy=> bAxisHomeBusy, 
	Active=> bAxisHomeActive, 
	CommandAborted=> bAxisHomeAborted, 
	Error=> bAxisHomeError, 
	ErrorID=> nAxisHomeErrorID);
	//Lefutás ellenőrzése
IF (bAxisHomeDone AND NOT(bAxisHomeBusy OR bAxisHomeActive OR bAxisHomeAborted OR bAxisHomeError)) THEN
	lrJozsiPosition:=GVL.lrNTCSzervizbox;
	sJozsiAxisCommand := 'MOVE';
	bHomeReady:=TRUE;
END_IF
	
	//Move
fbJozsiMoveAbsolute(
	Axis:= GVL.axisJozsiTengely, 
	Execute:= sJozsiAxisCommand='MOVE' AND bJozsiTengelySzabad_TON.Q AND bHomeReady, 
	Position:= lrJozsiPosition, // -1115...0
	Velocity:= 1000, 
	Acceleration:= 0, 
	Deceleration:= 0, 
	Jerk:= 0, 
	BufferMode:= , 
	Options:= , 
	Done=> bAxisMoveDone, 
	Busy=> bAxisMoveBusy, 
	Active=> bAxisMoveActive, 
	CommandAborted=> bAxisMoveAborted, 
	Error=> bAxisMoveError, 
	ErrorID=> nAxisMoveErrorID);
	//Lefutás ellenőrzése
IF (bAxisMoveDone AND NOT(bAxisMoveBusy OR bAxisMoveActive OR bAxisMoveAborted OR bAxisMoveError)) THEN
	sJozsiAxisCommand := '';
END_IF
	
	//JOG
	fbJozsitengelyJOG(
	Axis:= GVL.axisJozsiTengely, 
	JogForward:= bJozsiJOGPlus AND bJozsiTengelySzabad_TON.Q, 
	JogBackwards:= bJozsiJOGMinus AND bJozsiTengelySzabad_TON.Q, 
	Mode:= MC_JOGMODE_STANDARD_SLOW, 
	Position:= , 
	Velocity:= 100, 
	Acceleration:= 0, 
	Deceleration:= 0, 
	Jerk:= 0, 
	Done=> bAxisCommandDone, 
	Busy=> bAxisCommandBusy, 
	Active=> bAxisCommandActive, 
	CommandAborted=> bAxisCommandAborted, 
	Error=> bAxisCommandError, 
	ErrorID=> nAxisCommandErrorID);
	
	//RESET ERROR
	fbJozsitengelyReset(
	Axis:= GVL.axisJozsiTengely, 
	Execute:= bJozsiReset, 
	Done=> bAxisCommandDone, 
	Busy=> bAxisCommandBusy, 
	Error=> bAxisCommandError, 
	ErrorID=> nAxisCommandErrorID);
	
	//Ha nem szabad futtatni
//	IF(NOT(bJozsiTengelySzabad)) THEN
//		sJozsiAxisCommand:='!INTERRUPTED';
//	END_IF

END_PROGRAM

// ---- POUs/GENERAL/Helpers/f_RobotNTCTengelytolTavol.TcPOU
FUNCTION f_RobotNTCTengelytolTavol : BOOL

f_RobotNTCTengelytolTavol:=(GVL.stRobotStatusz.rX>-100) 
							OR (GVL.stRobotStatusz.rY>350)
							OR (GVL.stRobotStatusz.rZ>-111);

END_FUNCTION

// ---- POUs/MAIN.TcPOU
PROGRAM MAIN
VAR_INPUT
	bLevego AT %Q*: BOOL := FALSE;	
END_VAR
VAR_OUTPUT
	bLevegoOK AT %I*: BOOL;	
END_VAR
VAR
	bZoliGomb AT %I* : BOOL;
	bZoliSzelep AT %Q*: BOOL := FALSE;

	bPartsReadReady: BOOL;	
	bSettingsReadReady: BOOL;	
	iInd: INT;
	bTypeFound: BOOL;

	iState: INT:=3;
	sPartsString: STRING;
	sPartsGetStr: T_MaxString;
	iStateS: INT:=3;
	sSettingsString: T_MaxString;
	sSettingsGetStr: T_MaxString;
	iEqu: INT;

	// Fájlnyitás
	bPartsOpenExecute: BOOL := FALSE;
	PartsOpen: fb_FileOpen;
	nPartsOpenMode: DWORD;
	bPartsOpenBusy: BOOL;
	bPartsOpenError: BOOL;
	nPartsOpenError: UDINT;
	hPartsFile: UINT;
	
	bSettingsOpenExecute: BOOL := FALSE;
	SettingsOpen: fb_FileOpen;
	nSettingsOpenMode: DWORD;
	bSettingsOpenBusy: BOOL;
	bSettingsOpenError: BOOL;
	nSettingsOpenError: UDINT;
	hSettingsFile: UINT;
	
	// Fájlírás
	PartsPutStr: fb_FilePuts;
	bPartsPutStrExecute: BOOL;
	bPartsPutStrBusy: BOOL;
	bPartsPutStrError: BOOL;
	nPartsPutStrError: UDINT;
	
	SettingsPutStr: fb_FilePuts;
	bSettingsPutStrExecute: BOOL;
	bSettingsPutStrBusy: BOOL;
	bSettingsPutStrError: BOOL;
	nSettingsPutStrError: UDINT;

	// Fájlolvasás
	PartsGetStr: fb_FileGets;
	bPartsGetStrExecute: BOOL;
	bPartsGetStrBusy: BOOL;
	bPartsGetStrError: BOOL;
	nPartsGetStrError: UDINT;

	SettingsGetStr: fb_FileGets;
	bSettingsGetStrExecute: BOOL;
	bSettingsGetStrBusy: BOOL;
	bSettingsGetStrError: BOOL;
	nSettingsGetStrError: UDINT;
	
	// Fájlzárás
	PartsClose: fb_FileClose;
	bPartsCloseExecute: BOOL;
	bPartsCloseBusy: BOOL;
	bPartsCloseError: BOOL;
	nPartsCloseError: UDINT;

	SettingsClose: fb_FileClose;
	bSettingsCloseExecute: BOOL;
	bSettingsCloseBusy: BOOL;
	bSettingsCloseError: BOOL;
	nSettingsCloseError: UDINT;

	bGetStrPartsEOF: BOOL;
	bGetStrSettingsEOF: BOOL;
	raParameters: ARRAY[0..25] OF REAL;
	Ind: INT;
	sParName: STRING;
	sParValue: STRING;
	sParLine: STRING;
	R_TRIG_BiztZar: R_TRIG;
	
	F_TRIG_BiztZar: F_TRIG;
	TON_Biztzar: TON;
	TON_Biztzar_Start: BOOL;
END_VAR

GVL.fbWritePersistentData(
						NETID:='10.0.0.31.1.1',
						PORT:=851,
						START:=GVL.bStart_WrPer,
						TMOUT:=T#1S,
						BUSY=>GVL.bBusy_WrPer,
						ERR=>GVL.bError_WrPer);


IF (NOT GVL.bBusy_WrPer OR GVL.bError_WrPer) AND GVL.bStart_WrPer THEN
	GVL.bStart_WrPer:=FALSE;
END_IF


IF bZoliGomb=TRUE THEN
	bZoliSzelep := TRUE;
ELSE
	bZoliSzelep := FALSE;
END_IF

TON_Biztzar(IN:=TON_Biztzar_Start, PT:=T#200MS);
R_TRIG_BiztZar(CLK:=GVL.bBiztonsagiZarGomb);
F_TRIG_BiztZar(CLK:=GVL.bBiztonsagiZarGomb);

IF F_TRIG_BiztZar.Q THEN
//	WHILE NOT (ROBOTREMOTE.sRobotCommand='') DO
//		;
//	END_WHILE
//	ROBOTREMOTE.sRobotCommand := 'Pause';
//	ROBOTREMOTE.bRobotCommandSend := TRUE;
	GVL.bBiztonsagiZarBe:=FALSE;
//
END_IF

IF R_TRIG_BiztZar.Q THEN
//	WHILE NOT (ROBOTREMOTE.sRobotCommand='') DO
//		;
//	END_WHILE
	GVL.bBiztonsagiZarBe:=TRUE;
	TON_Biztzar_Start:=TRUE;
//	ROBOTREMOTE.sRobotCommand := 'Continue';
//	ROBOTREMOTE.bRobotCommandSend := TRUE;
END_IF
IF TON_Biztzar.Q THEN
	ROBOTREMOTE.sRobotCommand := 'Continue';
	ROBOTREMOTE.bRobotCommandSend := TRUE;
	TON_Biztzar_Start:=FALSE;
END_IF


CASE iState OF
	2:	// Alkatrészváltozás figyelése
		IF NOT((GVL.sNTCType=GVL.sNTCTypeElozo)
			AND (GVL.sPtType=GVL.sPtTypeElozo)
			AND (GVL.sProductType=GVL.sProductTypeElozo)) THEN
			GVL.bProductTypeOK:=FALSE;	
			IF NOT(GVL.sNTCType=GVL.sNTCTypeElozo) THEN
				IF (LEN(GVL.sNTCType)=32) THEN
					GVL.sNTCType:=RIGHT(GVL.sNTCType,23);
					GVL.sNTCType:=LEFT(GVL.sNTCType,6);
					iState:=3;
				ELSE
					GVL.sNTCType:='HIBÁS KÓD';
				END_IF;
				GVL.sNTCTypeElozo:=GVL.sNTCType;
			END_IF;
			IF NOT(GVL.sPtType=GVL.sPtTypeElozo) THEN
				IF (LEN(GVL.sPtType)=32) THEN
					GVL.sPtType:=RIGHT(GVL.sPtType,23);
					GVL.sPtType:=LEFT(GVL.sPtType,6);
					iState:=3;
				ELSE
					GVL.sPtType:='HIBÁS KÓD';
				END_IF;
				GVL.sPtTypeElozo:=GVL.sPtType;
			END_IF;
			IF NOT(GVL.sProductType=GVL.sProductTypeElozo) THEN
				IF NOT ((GVL.sProductType='637900')
					OR (GVL.sProductType='637901')
					OR (GVL.sProductType='637910')
					OR (GVL.sProductType='637911')
					OR	(GVL.sProductType='637920')
					OR (GVL.sProductType='637921')
					OR (GVL.sProductType='637930')
					OR (GVL.sProductType='637931')
					OR (GVL.sProductType='745900')
					OR (GVL.sProductType='745905')
					OR (GVL.sProductType='745906')
					OR (GVL.sProductType='745907')
					OR (GVL.sProductType='745910')
					OR (GVL.sProductType='745915')
					OR (GVL.sProductType='745916')
					OR (GVL.sProductType='745917')
					OR	(GVL.sProductType='521950')) THEN
					GVL.sProductType:='HIBÁS KÓD';
					GVL.iSelectedProductType:=-1;					
				END_IF
				GVL.sProductTypeElozo:=GVL.sProductType;
			END_IF;
			GVL.bProductTypeOK:=
			(((GVL.sProductType='637900') OR (GVL.sProductType='637901') OR (GVL.sProductType='745900') OR (GVL.sProductType='745910'))
				AND ((GVL.sNTCType='567604') OR (GVL.sNTCType='637707')) AND (GVL.sPtType='637710'))
			OR	(((GVL.sProductType='637910') OR (GVL.sProductType='637911') OR (GVL.sProductType='745905') OR (GVL.sProductType='745915'))
				AND ((GVL.sNTCType='567604') OR (GVL.sNTCType='637707')) AND (GVL.sPtType='637711'))
			OR	(((GVL.sProductType='637920') OR (GVL.sProductType='637921') OR (GVL.sProductType='745907') OR (GVL.sProductType='745917'))
				AND ((GVL.sNTCType='509647') OR (GVL.sNTCType='637700')) AND (GVL.sPtType='637710'))
			OR	(((GVL.sProductType='637930') OR (GVL.sProductType='637931') OR (GVL.sProductType='745906') OR (GVL.sProductType='745916'))
				AND ((GVL.sNTCType='509647') OR (GVL.sNTCType='637700')) AND (GVL.sPtType='637711'))
			OR	(GVL.sProductType='521950');
			IF GVL.bProductTypeOK=TRUE THEN
				bTypeFound:=FALSE;
				iInd:=0;
				WHILE (NOT bTypeFound) AND (iInd<11) DO
					IF GVL.sProductType=GVL.saProductTypes[iInd] THEN
						bTypeFound:=TRUE;
						GVL.iSelectedProductType:=iInd; // Ezzel kezdeményezzük a termékváltást
					ELSE
						iInd:=iInd+1;
					END_IF
				END_WHILE
				IF GVL.iSelectedProductType=8 THEN
					Laser.s_InCommand:='SETJOB_521';
				ELSIF GVL.iSelectedProductType<8 THEN
					Laser.s_InCommand:='SETJOB_637';
					GVL.bKameraPROG:=FALSE;
					GVL.nWeldingStopDistance1:=GVL.nWeldingStopDistance1_637;
					GVL.nWeldingStopDistance2:=GVL.nWeldingStopDistance2_637;
					GVL.nWeldingStopDistance3:=GVL.nWeldingStopDistance3_637;
					GVL.nWeldingStopDistance4:=GVL.nWeldingStopDistance4_637;
					GVL.nWeldingStopDistance5:=GVL.nWeldingStopDistance5_637;
					GVL.nWeldingDistanceMin1:=GVL.nWeldingDistanceMin1_637;
					GVL.nWeldingDistanceMin2:=GVL.nWeldingDistanceMin2_637;
					GVL.nWeldingDistanceMin3:=GVL.nWeldingDistanceMin3_637;
					GVL.nWeldingDistanceMin4:=GVL.nWeldingDistanceMin4_637;
					GVL.nWeldingDistanceMin5:=GVL.nWeldingDistanceMin5_637;
					GVL.nWeldingDistanceMax1:=GVL.nWeldingDistanceMax1_637;
					GVL.nWeldingDistanceMax2:=GVL.nWeldingDistanceMax2_637;
					GVL.nWeldingDistanceMax3:=GVL.nWeldingDistanceMax3_637;
					GVL.nWeldingDistanceMax4:=GVL.nWeldingDistanceMax4_637;
					GVL.nWeldingDistanceMax5:=GVL.nWeldingDistanceMax5_637;
				ELSIF GVL.iSelectedProductType>8 THEN
					GVL.bKameraPROG:=TRUE;
					GVL.nWeldingStopDistance1:=GVL.nWeldingStopDistance1_745;
					GVL.nWeldingStopDistance2:=GVL.nWeldingStopDistance2_745;
					GVL.nWeldingStopDistance3:=GVL.nWeldingStopDistance3_745;
					GVL.nWeldingStopDistance4:=GVL.nWeldingStopDistance4_745;
					GVL.nWeldingStopDistance5:=GVL.nWeldingStopDistance5_745;
					GVL.nWeldingDistanceMin1:=GVL.nWeldingDistanceMin1_745;
					GVL.nWeldingDistanceMin2:=GVL.nWeldingDistanceMin2_745;
					GVL.nWeldingDistanceMin3:=GVL.nWeldingDistanceMin3_745;
					GVL.nWeldingDistanceMin4:=GVL.nWeldingDistanceMin4_745;
					GVL.nWeldingDistanceMin5:=GVL.nWeldingDistanceMin5_745;
					GVL.nWeldingDistanceMax1:=GVL.nWeldingDistanceMax1_745;
					GVL.nWeldingDistanceMax2:=GVL.nWeldingDistanceMax2_745;
					GVL.nWeldingDistanceMax3:=GVL.nWeldingDistanceMax3_745;
					GVL.nWeldingDistanceMax4:=GVL.nWeldingDistanceMax4_745;
					GVL.nWeldingDistanceMax5:=GVL.nWeldingDistanceMax5_745;
					IF GVL.iSelectedProductType>8 AND GVL.iSelectedProductType MOD 2=1 THEN // 74590X
						Laser.s_InCommand:='SETJOB_745900';
					ELSIF GVL.iSelectedProductType>8 AND GVL.iSelectedProductType MOD 2=0 THEN // 74591X
						Laser.s_InCommand:='SETJOB_745910';
					END_IF
				END_IF
			END_IF
		END_IF
	3:	// "Parts" fájl megnyitásának kezdeményezése
		bPartsOpenExecute:=TRUE;
		IF bPartsReadReady=TRUE THEN
			nPartsOpenMode:=FOPEN_MODETEXT OR FOPEN_MODEWRITE;
		ELSE
			nPartsOpenMode:=FOPEN_MODETEXT OR FOPEN_MODEREAD;
		END_IF;
		iState:=4;
	4:	// Várakozás a busy jelre
		IF bPartsOpenBusy=TRUE THEN
			iState:=5;
		END_IF
	5:	// Várakozás a fájlnyitás befejeztére
		IF bPartsOpenBusy=FALSE THEN
			bPartsOpenExecute:=FALSE;
			IF bPartsReadReady=TRUE THEN
				iState:=6;
			ELSE
				iState:=26;
			END_IF
		END_IF
	6:	// Fájlnyitás sikerességének vizsgálata
		IF bPartsOpenError=FALSE THEN
			sPartsString:=CONCAT('NTC=',
							CONCAT(GVL.sNTCType,
							CONCAT('$R$N',
							CONCAT('PT1000=',GVL.sPtType))));
			iState:=7;
		ELSE
			iState:=101;
		END_IF
	7:	// Parts fájlba írás kezdeményezése
		bPartsPutStrExecute:=TRUE;
		iState:=8;
	8:	// Várakozás a busy jelre
		IF bPartsPutStrBusy=TRUE THEN
			iState:=9;
		END_IF
	9:	// Várakozás a fájlírás befejeztére
		IF bPartsPutStrBusy=FALSE THEN
			bPartsPutStrExecute:=FALSE;
			iState:=10;
		END_IF
	10:	// Fájlírás sikerességének vizsgálata
		IF bPartsPutStrError=FALSE THEN
			iState:=11;
		ELSE
			iState:=103;
		END_IF
	26:	// Fájlnyitás sikerességének vizsgálata
		IF bPartsOpenError=FALSE THEN
			iState:=27;
		ELSE
			iState:=101;
		END_IF
	27:	// Parts fájlból olvasás kezdeményezése
		bPartsGetStrExecute:=TRUE;
		iState:=28;
	28:	// Várakozás a busy jelre
		IF bPartsGetStrBusy=TRUE THEN
			iState:=29;
		END_IF
	29:	// Várakozás a fájlolvasás befejeztére
		IF bPartsGetStrBusy=FALSE THEN
			bPartsGetStrExecute:=FALSE;
			iState:=30;
		END_IF
	30:	// Fájlolvasás sikerességének vizsgálata
		IF bPartsGetStrError=FALSE THEN
			IF FIND(sPartsGetStr,'NTC')>0 THEN
				GVL.sNTCType:=LEFT(RIGHT(sPartsGetStr,LEN(sPartsGetStr)-FIND(sPartsGetStr,'=')),6);
				GVL.sNTCTypeElozo:=GVL.sNTCType;
			ELSIF FIND(sPartsGetStr,'PT1000')>0 THEN
				GVL.sPtType:=LEFT(RIGHT(sPartsGetStr,LEN(sPartsGetStr)-FIND(sPartsGetStr,'=')),6);
				GVL.sPtTypeElozo:=GVL.sPtType;
			END_IF
			IF bGetStrPartsEOF=FALSE THEN
				iState:=27;
			ELSE
				iState:=11;
			END_IF
		ELSE
			iState:=103;
		END_IF
	11:	// Parts fájl zárásának kezdeményezése
		bPartsCloseExecute:=TRUE;
		iState:=12;
	12:	// Várakozás a busy jelre
		IF bPartsCloseBusy=TRUE THEN
			iState:=13;
		END_IF
	13:	// Várakozás a fájlzárás befejeztére
		IF bPartsCloseBusy=FALSE THEN
			bPartsCloseExecute:=FALSE;
			iState:=14;
		END_IF
	14:	// Fájlzárás sikerességének vizsgálata
		IF bPartsCloseError=FALSE THEN
			bPartsReadReady:=TRUE;	
			iState:=2;
		ELSE
			iState:=104;
		END_IF
END_CASE

CASE iStateS OF
	2:	// Paraméterváltozás figyelése
		IF (GVL.bSettingsAutoSave=TRUE) AND
			NOT((GVL.bSettingsAutoSave=GVL.bSettingsAutoSaveElozo)
			AND (GVL.rNTCDev=GVL.rNTCDevElozo)
			AND (GVL.rNTC2Dev=GVL.rNTC2DevElozo)
			AND (GVL.rPtDev=GVL.rPtDevElozo)
			AND (GVL.rISOL_MAX=GVL.rISOL_MAXElozo)
			AND (GVL.rTempMax=GVL.rTempMaxElozo)
			AND (GVL.rIdoallandoMax=GVL.rIdoallandoMaxElozo)
			AND (GVL.PTRES_SOKK_MAX=GVL.PTRES_SOKK_MAXElozo)
			AND (GVL.lrPtSzervizbox=GVL.lrPtSzervizboxElozo)
			AND (GVL.lrHegesztoPosition6=GVL.lrHegesztoPosition6Elozo)
			AND (GVL.lrHegesztoPosition7=GVL.lrHegesztoPosition7Elozo)
			AND (GVL.lrRobotKappePosition=GVL.lrRobotKappePositionElozo)
			AND (GVL.lrKappePosition=GVL.lrKappePositionElozo)
			AND (GVL.lrKodolvasasPosition=GVL.lrKodolvasasPositionElozo)
			AND (GVL.lrKodolvasasPosition2=GVL.lrKodolvasasPosition2Elozo)
			AND (GVL.lrVegmeroPosition=GVL.lrVegmeroPositionElozo)
			AND (GVL.lrNTCSzervizbox=GVL.lrNTCSzervizboxElozo)
			AND (GVL.lrHajlitoPosition1=GVL.lrHajlitoPosition1Elozo)
			AND (GVL.lrHajlitoPosition2=GVL.lrHajlitoPosition2Elozo)
			AND (GVL.lrHegesztoPosition1=GVL.lrHegesztoPosition1Elozo)
			AND (GVL.lrHegesztoPosition2=GVL.lrHegesztoPosition2Elozo)
			AND (GVL.lrHegesztoPosition3=GVL.lrHegesztoPosition3Elozo)
			AND (GVL.lrHegesztoPosition4=GVL.lrHegesztoPosition4Elozo)
			AND (GVL.lrHegesztoPosition5=GVL.lrHegesztoPosition5Elozo)
			AND (GVL.nWeldingStopDistance1=GVL.nWeldingStopDistance1Elozo)
			AND (GVL.nWeldingStopDistance2=GVL.nWeldingStopDistance2Elozo)
			AND (GVL.nWeldingStopDistance3=GVL.nWeldingStopDistance3Elozo)
			AND (GVL.nWeldingStopDistance4=GVL.nWeldingStopDistance4Elozo)
			AND (GVL.nWeldingStopDistance5=GVL.nWeldingStopDistance5Elozo)
			AND (GVL.bAutomaticWeldingStop1=GVL.bAutomaticWeldingStop1Elozo)
			AND (GVL.bAutomaticWeldingStop2=GVL.bAutomaticWeldingStop2Elozo)
			AND (GVL.bAutomaticWeldingStop3=GVL.bAutomaticWeldingStop3Elozo)
			AND (GVL.bAutomaticWeldingStop4=GVL.bAutomaticWeldingStop4Elozo)
			AND (GVL.bAutomaticWeldingStop5=GVL.bAutomaticWeldingStop5Elozo)
			AND (GVL.nWeldingDistanceMin1=GVL.nWeldingDistanceMin1Elozo)
			AND (GVL.nWeldingDistanceMin2=GVL.nWeldingDistanceMin2Elozo)
			AND (GVL.nWeldingDistanceMin3=GVL.nWeldingDistanceMin3Elozo)
			AND (GVL.nWeldingDistanceMin4=GVL.nWeldingDistanceMin4Elozo)
			AND (GVL.nWeldingDistanceMin5=GVL.nWeldingDistanceMin5Elozo)
			AND (GVL.nWeldingDistanceMax1=GVL.nWeldingDistanceMax1Elozo)
			AND (GVL.nWeldingDistanceMax2=GVL.nWeldingDistanceMax2Elozo)
			AND (GVL.nWeldingDistanceMax3=GVL.nWeldingDistanceMax3Elozo)
			AND (GVL.nWeldingDistanceMax4=GVL.nWeldingDistanceMax4Elozo)
			AND (GVL.nWeldingDistanceMax5=GVL.nWeldingDistanceMax5Elozo)
			AND (GVL.lrNTCKameraPosition=GVL.lrNTCKameraPositionElozo)
			AND (GVL.lrPtKameraPosition=GVL.lrPtKameraPositionElozo)
			AND (GVL.nWeldingDistanceStartMin1=GVL.nWeldingDistanceStartMin1Elozo)
			AND (GVL.nWeldingDistanceStartMin2=GVL.nWeldingDistanceStartMin2Elozo)
			AND (GVL.nWeldingDistanceStartMin3=GVL.nWeldingDistanceStartMin3Elozo)
			AND (GVL.nWeldingDistanceStartMin4=GVL.nWeldingDistanceStartMin4Elozo)
			AND (GVL.nWeldingDistanceStartMin5=GVL.nWeldingDistanceStartMin5Elozo)
			AND (GVL.nWeldingDistanceStartMax1=GVL.nWeldingDistanceStartMax1Elozo)
			AND (GVL.nWeldingDistanceStartMax2=GVL.nWeldingDistanceStartMax2Elozo)
			AND (GVL.nWeldingDistanceStartMax3=GVL.nWeldingDistanceStartMax3Elozo)
			AND (GVL.nWeldingDistanceStartMax4=GVL.nWeldingDistanceStartMax4Elozo)
			AND (GVL.nWeldingDistanceStartMax5=GVL.nWeldingDistanceStartMax5Elozo)
			AND (GVL.lrCsiszoloPosition1=GVL.lrCsiszoloPosition1Elozo)
			AND (GVL.lrCsiszoloPosition2=GVL.lrCsiszoloPosition2Elozo)
			AND (GVL.nElectrode1Usage=GVL.nElectrode1UsageElozo)
			AND (GVL.nElectrode1UsageMax=GVL.nElectrode1UsageMaxElozo)
			AND (GVL.nElectrode1UsageWarn=GVL.nElectrode1UsageWarnElozo)
			AND (GVL.nElectrode2Usage=GVL.nElectrode2UsageElozo)
			AND (GVL.nElectrode2UsageMax=GVL.nElectrode2UsageMaxElozo)
			AND (GVL.nElectrode2UsageWarn=GVL.nElectrode2UsageWarnElozo)
			AND (GVL.nElectrode3Usage=GVL.nElectrode3UsageElozo)
			AND (GVL.nElectrode3UsageWarn=GVL.nElectrode3UsageWarnElozo)
			AND (GVL.nElectrode3UsageMax=GVL.nElectrode3UsageMaxElozo)
			AND (GVL.nHegFejTisztCiklusok=GVL.nHegFejTisztCiklusokElozo)
			AND (GVL.nHegFejTisztProgram=GVL.nHegFejTisztProgramElozo)
			AND (GVL.bWeldingLog=GVL.bWeldingLogElozo)) THEN
			iStateS:=3;
		END_IF
	3:	// "Parts" fájl megnyitásának kezdeményezése
		bSettingsOpenExecute:=TRUE;
		IF bSettingsReadReady=TRUE THEN
			nSettingsOpenMode:=FOPEN_MODETEXT OR FOPEN_MODEWRITE;
		ELSE
			nSettingsOpenMode:=FOPEN_MODETEXT OR FOPEN_MODEREAD;
		END_IF;
		iStateS:=4;
	4:	// Várakozás a busy jelre
		IF bSettingsOpenBusy=TRUE THEN
			iStateS:=5;
		END_IF
	5:	// Várakozás a fájlnyitás befejeztére
		IF bSettingsOpenBusy=FALSE THEN
			bSettingsOpenExecute:=FALSE;
			IF bSettingsReadReady=TRUE THEN
				iStateS:=6;
			ELSE
				iStateS:=26;
			END_IF
		END_IF
	6:	// Fájlnyitás sikerességének vizsgálata
		IF bSettingsOpenError=FALSE THEN
			Ind:=0;
			sSettingsString:='';
			iStateS:=7;
		ELSE
			iStateS:=101;
		END_IF
	7:	// Hegesztési információk mentésének előkészítése termékspecifikusan
		IF GVL.iSelectedProductType<8 THEN
			GVL.nWeldingStopDistance1_637:=GVL.nWeldingStopDistance1;
			GVL.nWeldingStopDistance2_637:=GVL.nWeldingStopDistance2;
			GVL.nWeldingStopDistance3_637:=GVL.nWeldingStopDistance3;
			GVL.nWeldingStopDistance4_637:=GVL.nWeldingStopDistance4;
			GVL.nWeldingStopDistance5_637:=GVL.nWeldingStopDistance5;
			GVL.nWeldingDistanceMin1_637:=GVL.nWeldingDistanceMin1;
			GVL.nWeldingDistanceMin2_637:=GVL.nWeldingDistanceMin2;
			GVL.nWeldingDistanceMin3_637:=GVL.nWeldingDistanceMin3;
			GVL.nWeldingDistanceMin4_637:=GVL.nWeldingDistanceMin4;
			GVL.nWeldingDistanceMin5_637:=GVL.nWeldingDistanceMin5;
			GVL.nWeldingDistanceMax1_637:=GVL.nWeldingDistanceMax1;
			GVL.nWeldingDistanceMax2_637:=GVL.nWeldingDistanceMax2;
			GVL.nWeldingDistanceMax3_637:=GVL.nWeldingDistanceMax3;
			GVL.nWeldingDistanceMax4_637:=GVL.nWeldingDistanceMax4;
			GVL.nWeldingDistanceMax5_637:=GVL.nWeldingDistanceMax5;
		ELSIF GVL.iSelectedProductType>8 THEN
			GVL.nWeldingStopDistance1_745:=GVL.nWeldingStopDistance1;
			GVL.nWeldingStopDistance2_745:=GVL.nWeldingStopDistance2;
			GVL.nWeldingStopDistance3_745:=GVL.nWeldingStopDistance3;
			GVL.nWeldingStopDistance4_745:=GVL.nWeldingStopDistance4;
			GVL.nWeldingStopDistance5_745:=GVL.nWeldingStopDistance5;
			GVL.nWeldingDistanceMin1_745:=GVL.nWeldingDistanceMin1;
			GVL.nWeldingDistanceMin2_745:=GVL.nWeldingDistanceMin2;
			GVL.nWeldingDistanceMin3_745:=GVL.nWeldingDistanceMin3;
			GVL.nWeldingDistanceMin4_745:=GVL.nWeldingDistanceMin4;
			GVL.nWeldingDistanceMin5_745:=GVL.nWeldingDistanceMin5;
			GVL.nWeldingDistanceMax1_745:=GVL.nWeldingDistanceMax1;
			GVL.nWeldingDistanceMax2_745:=GVL.nWeldingDistanceMax2;
			GVL.nWeldingDistanceMax3_745:=GVL.nWeldingDistanceMax3;
			GVL.nWeldingDistanceMax4_745:=GVL.nWeldingDistanceMax4;
			GVL.nWeldingDistanceMax5_745:=GVL.nWeldingDistanceMax5;
		END_IF
		iStateS:=8;
	8:	// Soronkövetkező sor és mentendő STRING előállítása
		CASE Ind OF
			0: sParName:='AUTOSAVE'; sParValue:=BOOL_TO_STRING(GVL.bSettingsAutoSave);
			1: sParName:='NTCTOL'; sParValue:=REAL_TO_STRING(GVL.rNTCDev);
			2: sParName:='NTC2TOL'; sParValue:=REAL_TO_STRING(GVL.rNTC2Dev);
			3: sParName:='PTTOL'; sParValue:=REAL_TO_STRING(GVL.rPtDev);
			4: sParName:='SZIGMAX'; sParValue:=REAL_TO_STRING(GVL.rISOL_MAX);
			5: sParName:='TOMBHOM'; sParValue:=REAL_TO_STRING(GVL.rTempMax);
			6: sParName:='IDOALLMAX'; sParValue:=REAL_TO_STRING(GVL.rIdoallandoMax);
			7: sParName:='SOKKMAX'; sParValue:=REAL_TO_STRING(GVL.PTRES_SOKK_MAX);
			8: sParName:='PTSZERVPOZ'; sParValue:=LREAL_TO_STRING(GVL.lrPtSzervizbox);
			9: sParName:='HEG6POZ'; sParValue:=LREAL_TO_STRING(GVL.lrHegesztoPosition6);
			10: sParName:='HEG7POZ'; sParValue:=LREAL_TO_STRING(GVL.lrHegesztoPosition7);
			11: sParName:='ROBKAPPOZ'; sParValue:=LREAL_TO_STRING(GVL.lrRobotKappePosition);
			12: sParName:='KAPPOZ'; sParValue:=LREAL_TO_STRING(GVL.lrKappePosition);
			13: sParName:='KODPOZ'; sParValue:=LREAL_TO_STRING(GVL.lrKodolvasasPosition);
			14: sParName:='KODPOZ2'; sParValue:=LREAL_TO_STRING(GVL.lrKodolvasasPosition2);
			15: sParName:='VEGMEROPOZ'; sParValue:=LREAL_TO_STRING(GVL.lrVegmeroPosition);
			16: sParName:='NTCSZERVPOZ'; sParValue:=LREAL_TO_STRING(GVL.lrNTCSzervizbox);
			17: sParName:='HAJL1POZ'; sParValue:=LREAL_TO_STRING(GVL.lrHajlitoPosition1);
			18: sParName:='HAJL2POZ'; sParValue:=LREAL_TO_STRING(GVL.lrHajlitoPosition2);
			19: sParName:='HEG1POZ'; sParValue:=LREAL_TO_STRING(GVL.lrHegesztoPosition1);
			20: sParName:='HEG2POZ'; sParValue:=LREAL_TO_STRING(GVL.lrHegesztoPosition2);
			21: sParName:='HEG3POZ'; sParValue:=LREAL_TO_STRING(GVL.lrHegesztoPosition3);
			22: sParName:='HEG4POZ'; sParValue:=LREAL_TO_STRING(GVL.lrHegesztoPosition4);
			23: sParName:='HEG5POZ'; sParValue:=LREAL_TO_STRING(GVL.lrHegesztoPosition5);
			24: sParName:='HEGSTOPTAV1'; sParValue:=DINT_TO_STRING(GVL.nWeldingStopDistance1_637);
			25: sParName:='HEGSTOPTAV2'; sParValue:=DINT_TO_STRING(GVL.nWeldingStopDistance2_637);
			26: sParName:='HEGSTOPTAV3'; sParValue:=DINT_TO_STRING(GVL.nWeldingStopDistance3_637);
			27: sParName:='HEGSTOPTAV4'; sParValue:=DINT_TO_STRING(GVL.nWeldingStopDistance4_637);
			28: sParName:='HEGSTOPTAV5'; sParValue:=DINT_TO_STRING(GVL.nWeldingStopDistance5_637);
			29: sParName:='HEGSTOPTAV1_2'; sParValue:=DINT_TO_STRING(GVL.nWeldingStopDistance1_745);
			30: sParName:='HEGSTOPTAV2_2'; sParValue:=DINT_TO_STRING(GVL.nWeldingStopDistance2_745);
			31: sParName:='HEGSTOPTAV3_2'; sParValue:=DINT_TO_STRING(GVL.nWeldingStopDistance3_745);
			32: sParName:='HEGSTOPTAV4_2'; sParValue:=DINT_TO_STRING(GVL.nWeldingStopDistance4_745);
			33: sParName:='HEGSTOPTAV5_2'; sParValue:=DINT_TO_STRING(GVL.nWeldingStopDistance5_745);
			34: sParName:='AUTHEGSTOP1'; sParValue:=BOOL_TO_STRING(GVL.bAutomaticWeldingStop1);
			35: sParName:='AUTHEGSTOP2'; sParValue:=BOOL_TO_STRING(GVL.bAutomaticWeldingStop2);
			36: sParName:='AUTHEGSTOP3'; sParValue:=BOOL_TO_STRING(GVL.bAutomaticWeldingStop3);
			37: sParName:='AUTHEGSTOP4'; sParValue:=BOOL_TO_STRING(GVL.bAutomaticWeldingStop4);
			38: sParName:='AUTHEGSTOP5'; sParValue:=BOOL_TO_STRING(GVL.bAutomaticWeldingStop5);
			39: sParName:='WELDINGLOG'; sParValue:=BOOL_TO_STRING(GVL.bWeldingLog);
			40: sParName:='HEGMINTAV1'; sParValue:=DINT_TO_STRING(GVL.nWeldingDistanceMin1_637);
			41: sParName:='HEGMINTAV2'; sParValue:=DINT_TO_STRING(GVL.nWeldingDistanceMin2_637);
			42: sParName:='HEGMINTAV3'; sParValue:=DINT_TO_STRING(GVL.nWeldingDistanceMin3_637);
			43: sParName:='HEGMINTAV4'; sParValue:=DINT_TO_STRING(GVL.nWeldingDistanceMin4_637);
			44: sParName:='HEGMINTAV5'; sParValue:=DINT_TO_STRING(GVL.nWeldingDistanceMin5_637);
			45: sParName:='HEGMINTAV1_2'; sParValue:=DINT_TO_STRING(GVL.nWeldingDistanceMin1_745);
			46: sParName:='HEGMINTAV2_2'; sParValue:=DINT_TO_STRING(GVL.nWeldingDistanceMin2_745);
			47: sParName:='HEGMINTAV3_2'; sParValue:=DINT_TO_STRING(GVL.nWeldingDistanceMin3_745);
			48: sParName:='HEGMINTAV4_2'; sParValue:=DINT_TO_STRING(GVL.nWeldingDistanceMin4_745);
			49: sParName:='HEGMINTAV5_2'; sParValue:=DINT_TO_STRING(GVL.nWeldingDistanceMin5_745);
			50: sParName:='HEGMAXTAV1'; sParValue:=DINT_TO_STRING(GVL.nWeldingDistanceMax1_637);
			51: sParName:='HEGMAXTAV2'; sParValue:=DINT_TO_STRING(GVL.nWeldingDistanceMax2_637);
			52: sParName:='HEGMAXTAV3'; sParValue:=DINT_TO_STRING(GVL.nWeldingDistanceMax3_637);
			53: sParName:='HEGMAXTAV4'; sParValue:=DINT_TO_STRING(GVL.nWeldingDistanceMax4_637);
			54: sParName:='HEGMAXTAV5'; sParValue:=DINT_TO_STRING(GVL.nWeldingDistanceMax5_637);
			55: sParName:='HEGMAXTAV1_2'; sParValue:=DINT_TO_STRING(GVL.nWeldingDistanceMax1_745);
			56: sParName:='HEGMAXTAV2_2'; sParValue:=DINT_TO_STRING(GVL.nWeldingDistanceMax2_745);
			57: sParName:='HEGMAXTAV3_2'; sParValue:=DINT_TO_STRING(GVL.nWeldingDistanceMax3_745);
			58: sParName:='HEGMAXTAV4_2'; sParValue:=DINT_TO_STRING(GVL.nWeldingDistanceMax4_745);
			59: sParName:='HEGMAXTAV5_2'; sParValue:=DINT_TO_STRING(GVL.nWeldingDistanceMax5_745);
			60: sParName:='NTCKAMPOZ'; sParValue:=LREAL_TO_STRING(GVL.lrNTCKameraPosition);
			61: sParName:='PTKAMPOZ'; sParValue:=LREAL_TO_STRING(GVL.lrPtKameraPosition);
			62: sParName:='HEGMINSTARTTAV1'; sParValue:=DINT_TO_STRING(GVL.nWeldingDistanceStartMin1);
			63: sParName:='HEGMINSTARTTAV2'; sParValue:=DINT_TO_STRING(GVL.nWeldingDistanceStartMin2);
			64: sParName:='HEGMINSTARTTAV3'; sParValue:=DINT_TO_STRING(GVL.nWeldingDistanceStartMin3);
			65: sParName:='HEGMINSTARTTAV4'; sParValue:=DINT_TO_STRING(GVL.nWeldingDistanceStartMin4);
			66: sParName:='HEGMINSTARTTAV5'; sParValue:=DINT_TO_STRING(GVL.nWeldingDistanceStartMin5);
			67: sParName:='HEGMAXSTARTTAV1'; sParValue:=DINT_TO_STRING(GVL.nWeldingDistanceStartMax1);
			68: sParName:='HEGMAXSTARTTAV2'; sParValue:=DINT_TO_STRING(GVL.nWeldingDistanceStartMax2);
			69: sParName:='HEGMAXSTARTTAV3'; sParValue:=DINT_TO_STRING(GVL.nWeldingDistanceStartMax3);
			70: sParName:='HEGMAXSTARTTAV4'; sParValue:=DINT_TO_STRING(GVL.nWeldingDistanceStartMax4);
			71: sParName:='HEGMAXSTARTTAV5'; sParValue:=DINT_TO_STRING(GVL.nWeldingDistanceStartMax5);
			72: sParName:='CSISZ1POZ'; sParValue:=LREAL_TO_STRING(GVL.lrCsiszoloPosition1);
			73: sParName:='CSISZ2POZ'; sParValue:=LREAL_TO_STRING(GVL.lrCsiszoloPosition2);
			74: sParName:='ELEKTRHASZ1'; sParValue:=DINT_TO_STRING(GVL.nElectrode1Usage);
			75: sParName:='ELEKTRHASZ1FIGY'; sParValue:=DINT_TO_STRING(GVL.nElectrode1UsageWarn);
			76: sParName:='ELEKTRHASZ1MAX'; sParValue:=DINT_TO_STRING(GVL.nElectrode1UsageMax);
			77: sParName:='ELEKTRHASZ2'; sParValue:=DINT_TO_STRING(GVL.nElectrode2Usage);
			78: sParName:='ELEKTRHASZ2FIGY'; sParValue:=DINT_TO_STRING(GVL.nElectrode2UsageWarn);
			79: sParName:='ELEKTRHASZ2MAX'; sParValue:=DINT_TO_STRING(GVL.nElectrode2UsageMax);
			80: sParName:='ELEKTRHASZ3'; sParValue:=DINT_TO_STRING(GVL.nElectrode3Usage);
			81: sParName:='ELEKTRHASZ3FIGY'; sParValue:=DINT_TO_STRING(GVL.nElectrode3UsageWarn);
			82: sParName:='ELEKTRHASZ3MAX'; sParValue:=DINT_TO_STRING(GVL.nElectrode3UsageMax);
			83: sParName:='ELEKTRTISZTCIKL'; sParValue:=DINT_TO_STRING(GVL.nHegFejTisztCiklusok);
			84: sParName:='ELEKTRTISZTPROG'; sParValue:=DINT_TO_STRING(GVL.nHegFejTisztProgram);
		END_CASE
		sParLine:=CONCAT(sParName,
					CONCAT('=',
					CONCAT(sParValue,'$R$N')));
		IF LEN(sSettingsString)+LEN(sParLine)<255 THEN
			sSettingsString:=CONCAT(sSettingsString,sParLine);
			Ind:=Ind+1;
			IF Ind>84 THEN
				iStateS:=9;
			END_IF
		ELSE
			iStateS:=9;
		END_IF
	9:	// Parts fájlba írás kezdeményezése
		bSettingsPutStrExecute:=TRUE;
		iStateS:=10;
	10:	// Várakozás a busy jelre
		IF bSettingsPutStrBusy=TRUE THEN
			iStateS:=11;
		END_IF
	11:	// Várakozás a fájlírás befejeztére
		IF bSettingsPutStrBusy=FALSE THEN
			bSettingsPutStrExecute:=FALSE;
			iStateS:=12;
		END_IF
	12:	// Fájlírás sikerességének vizsgálata
		IF bSettingsPutStrError=FALSE THEN
			sSettingsString:='';
			IF Ind<85 THEN
				iStateS:=8;
			ELSE
				GVL.bSettingsAutoSaveElozo:=GVL.bSettingsAutoSave;
				GVL.rNTCDevElozo:=GVL.rNTCDev;
				GVL.rNTC2DevElozo:=GVL.rNTC2Dev;
				GVL.rPtDevElozo:=GVL.rPtDev;
				GVL.rISOL_MAXElozo:=GVL.rISOL_MAX;
				GVL.rTempMaxElozo:=GVL.rTempMax;
				GVL.rIdoallandoMaxElozo:=GVL.rIdoallandoMax;
				GVL.PTRES_SOKK_MAXElozo:=GVL.PTRES_SOKK_MAX;
				GVL.lrPtSzervizboxElozo:=GVL.lrPtSzervizbox;
				GVL.lrHegesztoPosition6Elozo:=GVL.lrHegesztoPosition6;
				GVL.lrHegesztoPosition7Elozo:=GVL.lrHegesztoPosition7;
				GVL.lrRobotKappePositionElozo:=GVL.lrRobotKappePosition;
				GVL.lrKappePositionElozo:=GVL.lrKappePosition;
				GVL.lrKodolvasasPositionElozo:=GVL.lrKodolvasasPosition;
				GVL.lrKodolvasasPosition2Elozo:=GVL.lrKodolvasasPosition2;
				GVL.lrVegmeroPositionElozo:=GVL.lrVegmeroPosition;
				GVL.lrNTCSzervizboxElozo:=GVL.lrNTCSzervizbox;
				GVL.lrHajlitoPosition1Elozo:=GVL.lrHajlitoPosition1;
				GVL.lrHajlitoPosition2Elozo:=GVL.lrHajlitoPosition2;
				GVL.lrHegesztoPosition1Elozo:=GVL.lrHegesztoPosition1;
				GVL.lrHegesztoPosition2Elozo:=GVL.lrHegesztoPosition2;
				GVL.lrHegesztoPosition3Elozo:=GVL.lrHegesztoPosition3;
				GVL.lrHegesztoPosition4Elozo:=GVL.lrHegesztoPosition4;
				GVL.lrHegesztoPosition5Elozo:=GVL.lrHegesztoPosition5;
				GVL.nWeldingStopDistance1Elozo:=GVL.nWeldingStopDistance1;
				GVL.nWeldingStopDistance2Elozo:=GVL.nWeldingStopDistance2;
				GVL.nWeldingStopDistance3Elozo:=GVL.nWeldingStopDistance3;
				GVL.nWeldingStopDistance4Elozo:=GVL.nWeldingStopDistance4;
				GVL.nWeldingStopDistance5Elozo:=GVL.nWeldingStopDistance5;
				GVL.bAutomaticWeldingStop1Elozo:=GVL.bAutomaticWeldingStop1;
				GVL.bAutomaticWeldingStop2Elozo:=GVL.bAutomaticWeldingStop2;
				GVL.bAutomaticWeldingStop3Elozo:=GVL.bAutomaticWeldingStop3;
				GVL.bAutomaticWeldingStop4Elozo:=GVL.bAutomaticWeldingStop4;
				GVL.bAutomaticWeldingStop5Elozo:=GVL.bAutomaticWeldingStop5;
				GVL.bWeldingLogElozo:=GVL.bWeldingLog;
				GVL.nWeldingDistanceMin1Elozo:=GVL.nWeldingDistanceMin1;
				GVL.nWeldingDistanceMin2Elozo:=GVL.nWeldingDistanceMin2;
				GVL.nWeldingDistanceMin3Elozo:=GVL.nWeldingDistanceMin3;
				GVL.nWeldingDistanceMin4Elozo:=GVL.nWeldingDistanceMin4;
				GVL.nWeldingDistanceMin5Elozo:=GVL.nWeldingDistanceMin5;
				GVL.nWeldingDistanceMax1Elozo:=GVL.nWeldingDistanceMax1;
				GVL.nWeldingDistanceMax2Elozo:=GVL.nWeldingDistanceMax2;
				GVL.nWeldingDistanceMax3Elozo:=GVL.nWeldingDistanceMax3;
				GVL.nWeldingDistanceMax4Elozo:=GVL.nWeldingDistanceMax4;
				GVL.nWeldingDistanceMax5Elozo:=GVL.nWeldingDistanceMax5;
				GVL.lrNTCKameraPositionElozo:=GVL.lrNTCKameraPosition;
				GVL.lrPtKameraPositionElozo:=GVL.lrPtKameraPosition;
				GVL.nWeldingDistanceStartMin1Elozo:=GVL.nWeldingDistanceStartMin1;
				GVL.nWeldingDistanceStartMin2Elozo:=GVL.nWeldingDistanceStartMin2;
				GVL.nWeldingDistanceStartMin3Elozo:=GVL.nWeldingDistanceStartMin3;
				GVL.nWeldingDistanceStartMin4Elozo:=GVL.nWeldingDistanceStartMin4;
				GVL.nWeldingDistanceStartMin5Elozo:=GVL.nWeldingDistanceStartMin5;
				GVL.nWeldingDistanceStartMax1Elozo:=GVL.nWeldingDistanceStartMax1;
				GVL.nWeldingDistanceStartMax2Elozo:=GVL.nWeldingDistanceStartMax2;
				GVL.nWeldingDistanceStartMax3Elozo:=GVL.nWeldingDistanceStartMax3;
				GVL.nWeldingDistanceStartMax4Elozo:=GVL.nWeldingDistanceStartMax4;
				GVL.nWeldingDistanceStartMax5Elozo:=GVL.nWeldingDistanceStartMax5;
				GVL.lrCsiszoloPosition1Elozo:=GVL.lrCsiszoloPosition1;
				GVL.lrCsiszoloPosition2Elozo:=GVL.lrCsiszoloPosition2;
				GVL.nElectrode1UsageElozo:=GVL.nElectrode1Usage;
				GVL.nElectrode1UsageWarnElozo:=GVL.nElectrode1UsageWarn;
				GVL.nElectrode1UsageMaxElozo:=GVL.nElectrode1UsageMax;
				GVL.nElectrode2UsageElozo:=GVL.nElectrode2Usage;
				GVL.nElectrode2UsageWarnElozo:=GVL.nElectrode2UsageWarn;
				GVL.nElectrode2UsageMaxElozo:=GVL.nElectrode2UsageMax;
				GVL.nElectrode3UsageElozo:=GVL.nElectrode3Usage;
				GVL.nElectrode3UsageWarnElozo:=GVL.nElectrode3UsageWarn;
				GVL.nElectrode3UsageMaxElozo:=GVL.nElectrode3UsageMax;
				GVL.nHegFejTisztCiklusokElozo:=GVL.nHegFejTisztCiklusok;
				GVL.nHegFejTisztProgramElozo:=GVL.nHegFejTisztProgram;
				IF GVL.nElectrode1Usage>GVL.nElectrode1UsageMax THEN
					GVL.nElectrode1AlarmColor:=16#FFFF0000;
				ELSE
					GVL.nElectrode1AlarmColor:=16#FFFFFF00;
				END_IF
				IF GVL.nElectrode2Usage>GVL.nElectrode2UsageMax THEN
					GVL.nElectrode2AlarmColor:=16#FFFF0000;
				ELSE
					GVL.nElectrode2AlarmColor:=16#FFFFFF00;
				END_IF
				IF GVL.nElectrode3Usage>GVL.nElectrode3UsageMax THEN
					GVL.nElectrode3AlarmColor:=16#FFFF0000;
				ELSE
					GVL.nElectrode3AlarmColor:=16#FFFFFF00;
				END_IF
				iStateS:=13;
			END_IF
		ELSE
			iStateS:=103;
		END_IF
		
	26:	// Fájlnyitás sikerességének vizsgálata
		IF bSettingsOpenError=FALSE THEN
			iStateS:=27;
			Ind:=0;
		ELSE
			iStateS:=101;
		END_IF
	27:	// Parts fájlból olvasás kezdeményezése
		bSettingsGetStrExecute:=TRUE;
		iStateS:=28;
	28:	// Várakozás a busy jelre
		IF bSettingsGetStrBusy=TRUE THEN
			iStateS:=29;
		END_IF
	29:	// Várakozás a fájlolvasás befejeztére
		IF bSettingsGetStrBusy=FALSE THEN
			bSettingsGetStrExecute:=FALSE;
			iStateS:=30;
		END_IF
	30:	// Fájlolvasás sikerességének vizsgálata
		IF bSettingsGetStrError=FALSE THEN
			iEqu:=FIND(sSettingsGetStr,'=');
			sParName:=LEFT(sSettingsGetStr,iEqu-1);
			sParValue:=RIGHT(sSettingsGetStr,LEN(sSettingsGetStr)-iEqu);
			sParValue:=LEFT(sParValue,LEN(sParValue)-2);
			IF sParName='AUTOSAVE' THEN GVL.bSettingsAutoSave:=STRING_TO_BOOL(sParValue);
			ELSIF sParName='NTCTOL' THEN GVL.rNTCDev:=STRING_TO_REAL(sParValue);
			ELSIF sParName='NTC2TOL' THEN GVL.rNTC2Dev:=STRING_TO_REAL(sParValue);
			ELSIF sParName='PTTOL' THEN GVL.rPtDev:=STRING_TO_REAL(sParValue);
			ELSIF sParName='SZIGMAX' THEN GVL.rISOL_MAX:=STRING_TO_REAL(sParValue);
			ELSIF sParName='TOMBHOM' THEN GVL.rTempMax:=STRING_TO_REAL(sParValue);
			ELSIF sParName='IDOALLMAX' THEN GVL.rIdoallandoMax:=STRING_TO_REAL(sParValue);
			ELSIF sParName='SOKKMAX' THEN GVL.PTRES_SOKK_MAX:=STRING_TO_REAL(sParValue);
			ELSIF sParName='PTSZERVPOZ' THEN GVL.lrPtSzervizbox:=STRING_TO_LREAL(sParValue);
			ELSIF sParName='HEG6POZ' THEN GVL.lrHegesztoPosition6:=STRING_TO_LREAL(sParValue);
			ELSIF sParName='HEG7POZ' THEN GVL.lrHegesztoPosition7:=STRING_TO_LREAL(sParValue);
			ELSIF sParName='ROBKAPPOZ' THEN GVL.lrRobotKappePosition:=STRING_TO_LREAL(sParValue);
			ELSIF sParName='KAPPOZ' THEN GVL.lrKappePosition:=STRING_TO_LREAL(sParValue);
			ELSIF sParName='KODPOZ' THEN GVL.lrKodolvasasPosition:=STRING_TO_LREAL(sParValue);
			ELSIF sParName='KODPOZ2' THEN GVL.lrKodolvasasPosition2:=STRING_TO_LREAL(sParValue);
			ELSIF sParName='VEGMEROPOZ' THEN GVL.lrVegmeroPosition:=STRING_TO_LREAL(sParValue);
			ELSIF sParName='NTCSZERVPOZ' THEN GVL.lrNTCSzervizbox:=STRING_TO_LREAL(sParValue);
			ELSIF sParName='HAJL1POZ' THEN GVL.lrHajlitoPosition1:=STRING_TO_LREAL(sParValue);
			ELSIF sParName='HAJL2POZ' THEN GVL.lrHajlitoPosition2:=STRING_TO_LREAL(sParValue);
			ELSIF sParName='HEG1POZ' THEN GVL.lrHegesztoPosition1:=STRING_TO_LREAL(sParValue);
			ELSIF sParName='HEG2POZ' THEN GVL.lrHegesztoPosition2:=STRING_TO_LREAL(sParValue);
			ELSIF sParName='HEG3POZ' THEN GVL.lrHegesztoPosition3:=STRING_TO_LREAL(sParValue);
			ELSIF sParName='HEG4POZ' THEN GVL.lrHegesztoPosition4:=STRING_TO_LREAL(sParValue);
			ELSIF sParName='HEG5POZ' THEN GVL.lrHegesztoPosition5:=STRING_TO_LREAL(sParValue);
			ELSIF sParName='HEGSTOPTAV1' THEN GVL.nWeldingStopDistance1_637:=STRING_TO_DINT(sParValue);
			ELSIF sParName='HEGSTOPTAV2' THEN GVL.nWeldingStopDistance2_637:=STRING_TO_DINT(sParValue);
			ELSIF sParName='HEGSTOPTAV3' THEN GVL.nWeldingStopDistance3_637:=STRING_TO_DINT(sParValue);
			ELSIF sParName='HEGSTOPTAV4' THEN GVL.nWeldingStopDistance4_637:=STRING_TO_DINT(sParValue);
			ELSIF sParName='HEGSTOPTAV5' THEN GVL.nWeldingStopDistance5_637:=STRING_TO_DINT(sParValue);
			ELSIF sParName='HEGSTOPTAV1_2' THEN GVL.nWeldingStopDistance1_745:=STRING_TO_DINT(sParValue);
			ELSIF sParName='HEGSTOPTAV2_2' THEN GVL.nWeldingStopDistance2_745:=STRING_TO_DINT(sParValue);
			ELSIF sParName='HEGSTOPTAV3_2' THEN GVL.nWeldingStopDistance3_745:=STRING_TO_DINT(sParValue);
			ELSIF sParName='HEGSTOPTAV4_2' THEN GVL.nWeldingStopDistance4_745:=STRING_TO_DINT(sParValue);
			ELSIF sParName='HEGSTOPTAV5_2' THEN GVL.nWeldingStopDistance5_745:=STRING_TO_DINT(sParValue);
			ELSIF sParName='AUTHEGSTOP1' THEN GVL.bAutomaticWeldingStop1:=STRING_TO_BOOL(sParValue);
			ELSIF sParName='AUTHEGSTOP2' THEN GVL.bAutomaticWeldingStop2:=STRING_TO_BOOL(sParValue);
			ELSIF sParName='AUTHEGSTOP3' THEN GVL.bAutomaticWeldingStop3:=STRING_TO_BOOL(sParValue);
			ELSIF sParName='AUTHEGSTOP4' THEN GVL.bAutomaticWeldingStop4:=STRING_TO_BOOL(sParValue);
			ELSIF sParName='AUTHEGSTOP5' THEN GVL.bAutomaticWeldingStop5:=STRING_TO_BOOL(sParValue);
			ELSIF sParName='WELDINGLOG' THEN GVL.bWeldingLog:=STRING_TO_BOOL(sParValue);
			ELSIF sParName='HEGMINTAV1' THEN GVL.nWeldingDistanceMin1_637:=STRING_TO_DINT(sParValue);
			ELSIF sParName='HEGMINTAV2' THEN GVL.nWeldingDistanceMin2_637:=STRING_TO_DINT(sParValue);
			ELSIF sParName='HEGMINTAV3' THEN GVL.nWeldingDistanceMin3_637:=STRING_TO_DINT(sParValue);
			ELSIF sParName='HEGMINTAV4' THEN GVL.nWeldingDistanceMin4_637:=STRING_TO_DINT(sParValue);
			ELSIF sParName='HEGMINTAV5' THEN GVL.nWeldingDistanceMin5_637:=STRING_TO_DINT(sParValue);
			ELSIF sParName='HEGMINTAV1_2' THEN GVL.nWeldingDistanceMin1_745:=STRING_TO_DINT(sParValue);
			ELSIF sParName='HEGMINTAV2_2' THEN GVL.nWeldingDistanceMin2_745:=STRING_TO_DINT(sParValue);
			ELSIF sParName='HEGMINTAV3_2' THEN GVL.nWeldingDistanceMin3_745:=STRING_TO_DINT(sParValue);
			ELSIF sParName='HEGMINTAV4_2' THEN GVL.nWeldingDistanceMin4_745:=STRING_TO_DINT(sParValue);
			ELSIF sParName='HEGMINTAV5_2' THEN GVL.nWeldingDistanceMin5_745:=STRING_TO_DINT(sParValue);
			ELSIF sParName='HEGMAXTAV1' THEN GVL.nWeldingDistanceMax1_637:=STRING_TO_DINT(sParValue);
			ELSIF sParName='HEGMAXTAV2' THEN GVL.nWeldingDistanceMax2_637:=STRING_TO_DINT(sParValue);
			ELSIF sParName='HEGMAXTAV3' THEN GVL.nWeldingDistanceMax3_637:=STRING_TO_DINT(sParValue);
			ELSIF sParName='HEGMAXTAV4' THEN GVL.nWeldingDistanceMax4_637:=STRING_TO_DINT(sParValue);
			ELSIF sParName='HEGMAXTAV5' THEN GVL.nWeldingDistanceMax5_637:=STRING_TO_DINT(sParValue);
			ELSIF sParName='HEGMAXTAV1_2' THEN GVL.nWeldingDistanceMax1_745:=STRING_TO_DINT(sParValue);
			ELSIF sParName='HEGMAXTAV2_2' THEN GVL.nWeldingDistanceMax2_745:=STRING_TO_DINT(sParValue);
			ELSIF sParName='HEGMAXTAV3_2' THEN GVL.nWeldingDistanceMax3_745:=STRING_TO_DINT(sParValue);
			ELSIF sParName='HEGMAXTAV4_2' THEN GVL.nWeldingDistanceMax4_745:=STRING_TO_DINT(sParValue);
			ELSIF sParName='HEGMAXTAV5_2' THEN GVL.nWeldingDistanceMax5_745:=STRING_TO_DINT(sParValue);
			ELSIF sParName='NTCKAMPOZ' THEN GVL.lrNTCKameraPosition:=STRING_TO_LREAL(sParValue);
			ELSIF sParName='PTKAMPOZ' THEN GVL.lrPtKameraPosition:=STRING_TO_LREAL(sParValue);
			ELSIF sParName='HEGMINSTARTTAV1' THEN GVL.nWeldingDistanceStartMin1:=STRING_TO_DINT(sParValue);
			ELSIF sParName='HEGMINSTARTTAV2' THEN GVL.nWeldingDistanceStartMin2:=STRING_TO_DINT(sParValue);
			ELSIF sParName='HEGMINSTARTTAV3' THEN GVL.nWeldingDistanceStartMin3:=STRING_TO_DINT(sParValue);
			ELSIF sParName='HEGMINSTARTTAV4' THEN GVL.nWeldingDistanceStartMin4:=STRING_TO_DINT(sParValue);
			ELSIF sParName='HEGMINSTARTTAV5' THEN GVL.nWeldingDistanceStartMin5:=STRING_TO_DINT(sParValue);
			ELSIF sParName='HEGMAXSTARTTAV1' THEN GVL.nWeldingDistanceStartMax1:=STRING_TO_DINT(sParValue);
			ELSIF sParName='HEGMAXSTARTTAV2' THEN GVL.nWeldingDistanceStartMax2:=STRING_TO_DINT(sParValue);
			ELSIF sParName='HEGMAXSTARTTAV3' THEN GVL.nWeldingDistanceStartMax3:=STRING_TO_DINT(sParValue);
			ELSIF sParName='HEGMAXSTARTTAV4' THEN GVL.nWeldingDistanceStartMax4:=STRING_TO_DINT(sParValue);
			ELSIF sParName='HEGMAXSTARTTAV5' THEN GVL.nWeldingDistanceStartMax5:=STRING_TO_DINT(sParValue);
			ELSIF sParName='CSISZ1POZ' THEN GVL.lrCsiszoloPosition1:=STRING_TO_LREAL(sParValue);
			ELSIF sParName='CSISZ2POZ' THEN GVL.lrCsiszoloPosition2:=STRING_TO_LREAL(sParValue);
			ELSIF sParName='ELEKTRHASZ1' THEN GVL.nElectrode1Usage:=STRING_TO_DINT(sParValue);
			ELSIF sParName='ELEKTRHASZ1FIGY' THEN GVL.nElectrode1UsageWarn:=STRING_TO_DINT(sParValue);
			ELSIF sParName='ELEKTRHASZ1MAX' THEN GVL.nElectrode1UsageMax:=STRING_TO_DINT(sParValue);
			ELSIF sParName='ELEKTRHASZ2' THEN GVL.nElectrode2Usage:=STRING_TO_DINT(sParValue);
			ELSIF sParName='ELEKTRHASZ2FIGY' THEN GVL.nElectrode2UsageWarn:=STRING_TO_DINT(sParValue);
			ELSIF sParName='ELEKTRHASZ2MAX' THEN GVL.nElectrode2UsageMax:=STRING_TO_DINT(sParValue);
			ELSIF sParName='ELEKTRHASZ3' THEN GVL.nElectrode3Usage:=STRING_TO_DINT(sParValue);
			ELSIF sParName='ELEKTRHASZ3FIGY' THEN GVL.nElectrode3UsageWarn:=STRING_TO_DINT(sParValue);
			ELSIF sParName='ELEKTRHASZ3MAX' THEN GVL.nElectrode3UsageMax:=STRING_TO_DINT(sParValue);
			ELSIF sParName='ELEKTRTISZTCIKL' THEN GVL.nHegFejTisztCiklusok:=STRING_TO_UINT(sParValue);
			ELSIF sParName='ELEKTRTISZTPROG' THEN GVL.nHegFejTisztProgram:=STRING_TO_UINT(sParValue);
			END_IF
			IF bGetStrSettingsEOF=FALSE THEN
				iStateS:=27;
				Ind:=Ind+1;
			ELSE
				// Termékspecifikus hegesztési paraméterek kiválasztása
				IF GVL.iSelectedProductType<8 THEN
					GVL.nWeldingStopDistance1:=GVL.nWeldingStopDistance1_637;
					GVL.nWeldingStopDistance2:=GVL.nWeldingStopDistance2_637;
					GVL.nWeldingStopDistance3:=GVL.nWeldingStopDistance3_637;
					GVL.nWeldingStopDistance4:=GVL.nWeldingStopDistance4_637;
					GVL.nWeldingStopDistance5:=GVL.nWeldingStopDistance5_637;
					GVL.nWeldingDistanceMin1:=GVL.nWeldingDistanceMin1_637;
					GVL.nWeldingDistanceMin2:=GVL.nWeldingDistanceMin2_637;
					GVL.nWeldingDistanceMin3:=GVL.nWeldingDistanceMin3_637;
					GVL.nWeldingDistanceMin4:=GVL.nWeldingDistanceMin4_637;
					GVL.nWeldingDistanceMin5:=GVL.nWeldingDistanceMin5_637;
					GVL.nWeldingDistanceMax1:=GVL.nWeldingDistanceMax1_637;
					GVL.nWeldingDistanceMax2:=GVL.nWeldingDistanceMax2_637;
					GVL.nWeldingDistanceMax3:=GVL.nWeldingDistanceMax3_637;
					GVL.nWeldingDistanceMax4:=GVL.nWeldingDistanceMax4_637;
					GVL.nWeldingDistanceMax5:=GVL.nWeldingDistanceMax5_637;
				ELSIF GVL.iSelectedProductType>8 THEN
					GVL.nWeldingStopDistance1:=GVL.nWeldingStopDistance1_745;
					GVL.nWeldingStopDistance2:=GVL.nWeldingStopDistance2_745;
					GVL.nWeldingStopDistance3:=GVL.nWeldingStopDistance3_745;
					GVL.nWeldingStopDistance4:=GVL.nWeldingStopDistance4_745;
					GVL.nWeldingStopDistance5:=GVL.nWeldingStopDistance5_745;
					GVL.nWeldingDistanceMin1:=GVL.nWeldingDistanceMin1_745;
					GVL.nWeldingDistanceMin2:=GVL.nWeldingDistanceMin2_745;
					GVL.nWeldingDistanceMin3:=GVL.nWeldingDistanceMin3_745;
					GVL.nWeldingDistanceMin4:=GVL.nWeldingDistanceMin4_745;
					GVL.nWeldingDistanceMin5:=GVL.nWeldingDistanceMin5_745;
					GVL.nWeldingDistanceMax1:=GVL.nWeldingDistanceMax1_745;
					GVL.nWeldingDistanceMax2:=GVL.nWeldingDistanceMax2_745;
					GVL.nWeldingDistanceMax3:=GVL.nWeldingDistanceMax3_745;
					GVL.nWeldingDistanceMax4:=GVL.nWeldingDistanceMax4_745;
					GVL.nWeldingDistanceMax5:=GVL.nWeldingDistanceMax5_745;
				END_IF
				// Automatikusan mentendő paraméterek változásának törlése
				GVL.bSettingsAutoSaveElozo:=GVL.bSettingsAutoSave;
				GVL.rNTCDevElozo:=GVL.rNTCDev;
				GVL.rNTC2DevElozo:=GVL.rNTC2Dev;
				GVL.rPtDevElozo:=GVL.rPtDev;
				GVL.rISOL_MAXElozo:=GVL.rISOL_MAX;
				GVL.rTempMaxElozo:=GVL.rTempMax;
				GVL.rIdoallandoMaxElozo:=GVL.rIdoallandoMax;
				GVL.PTRES_SOKK_MAXElozo:=GVL.PTRES_SOKK_MAX;
				GVL.lrPtSzervizboxElozo:=GVL.lrPtSzervizbox;
				GVL.lrHegesztoPosition6Elozo:=GVL.lrHegesztoPosition6;
				GVL.lrHegesztoPosition7Elozo:=GVL.lrHegesztoPosition7;
				GVL.lrRobotKappePositionElozo:=GVL.lrRobotKappePosition;
				GVL.lrKappePositionElozo:=GVL.lrKappePosition;
				GVL.lrKodolvasasPositionElozo:=GVL.lrKodolvasasPosition;
				GVL.lrKodolvasasPosition2Elozo:=GVL.lrKodolvasasPosition2;
				GVL.lrVegmeroPositionElozo:=GVL.lrVegmeroPosition;
				GVL.lrNTCSzervizboxElozo:=GVL.lrNTCSzervizbox;
				GVL.lrHajlitoPosition1Elozo:=GVL.lrHajlitoPosition1;
				GVL.lrHajlitoPosition2Elozo:=GVL.lrHajlitoPosition2;
				GVL.lrHegesztoPosition1Elozo:=GVL.lrHegesztoPosition1;
				GVL.lrHegesztoPosition2Elozo:=GVL.lrHegesztoPosition2;
				GVL.lrHegesztoPosition3Elozo:=GVL.lrHegesztoPosition3;
				GVL.lrHegesztoPosition4Elozo:=GVL.lrHegesztoPosition4;
				GVL.lrHegesztoPosition5Elozo:=GVL.lrHegesztoPosition5;
				GVL.nWeldingStopDistance1Elozo:=GVL.nWeldingStopDistance1;
				GVL.nWeldingStopDistance2Elozo:=GVL.nWeldingStopDistance2;
				GVL.nWeldingStopDistance3Elozo:=GVL.nWeldingStopDistance3;
				GVL.nWeldingStopDistance4Elozo:=GVL.nWeldingStopDistance4;
				GVL.nWeldingStopDistance5Elozo:=GVL.nWeldingStopDistance5;
				GVL.bAutomaticWeldingStop1Elozo:=GVL.bAutomaticWeldingStop1;
				GVL.bAutomaticWeldingStop2Elozo:=GVL.bAutomaticWeldingStop2;
				GVL.bAutomaticWeldingStop3Elozo:=GVL.bAutomaticWeldingStop3;
				GVL.bAutomaticWeldingStop4Elozo:=GVL.bAutomaticWeldingStop4;
				GVL.bAutomaticWeldingStop5Elozo:=GVL.bAutomaticWeldingStop5;
				GVL.bWeldingLogElozo:=GVL.bWeldingLog;
				GVL.nWeldingDistanceMin1Elozo:=GVL.nWeldingDistanceMin1;
				GVL.nWeldingDistanceMin2Elozo:=GVL.nWeldingDistanceMin2;
				GVL.nWeldingDistanceMin3Elozo:=GVL.nWeldingDistanceMin3;
				GVL.nWeldingDistanceMin4Elozo:=GVL.nWeldingDistanceMin4;
				GVL.nWeldingDistanceMin5Elozo:=GVL.nWeldingDistanceMin5;
				GVL.nWeldingDistanceMax1Elozo:=GVL.nWeldingDistanceMax1;
				GVL.nWeldingDistanceMax2Elozo:=GVL.nWeldingDistanceMax2;
				GVL.nWeldingDistanceMax3Elozo:=GVL.nWeldingDistanceMax3;
				GVL.nWeldingDistanceMax4Elozo:=GVL.nWeldingDistanceMax4;
				GVL.nWeldingDistanceMax5Elozo:=GVL.nWeldingDistanceMax5;
				GVL.lrNTCKameraPositionElozo:=GVL.lrNTCKameraPosition;
				GVL.lrPtKameraPositionElozo:=GVL.lrPtKameraPosition;
				GVL.nWeldingDistanceStartMin1Elozo:=GVL.nWeldingDistanceStartMin1;
				GVL.nWeldingDistanceStartMin2Elozo:=GVL.nWeldingDistanceStartMin2;
				GVL.nWeldingDistanceStartMin3Elozo:=GVL.nWeldingDistanceStartMin3;
				GVL.nWeldingDistanceStartMin4Elozo:=GVL.nWeldingDistanceStartMin4;
				GVL.nWeldingDistanceStartMin5Elozo:=GVL.nWeldingDistanceStartMin5;
				GVL.nWeldingDistanceStartMax1Elozo:=GVL.nWeldingDistanceStartMax1;
				GVL.nWeldingDistanceStartMax2Elozo:=GVL.nWeldingDistanceStartMax2;
				GVL.nWeldingDistanceStartMax3Elozo:=GVL.nWeldingDistanceStartMax3;
				GVL.nWeldingDistanceStartMax4Elozo:=GVL.nWeldingDistanceStartMax4;
				GVL.nWeldingDistanceStartMax5Elozo:=GVL.nWeldingDistanceStartMax5;
				GVL.lrCsiszoloPosition1Elozo:=GVL.lrCsiszoloPosition1;
				GVL.lrCsiszoloPosition2Elozo:=GVL.lrCsiszoloPosition2;
				GVL.nElectrode1UsageElozo:=GVL.nElectrode1Usage;
				GVL.nElectrode1UsageWarnElozo:=GVL.nElectrode1UsageWarn;
				GVL.nElectrode1UsageMaxElozo:=GVL.nElectrode1UsageMax;
				GVL.nElectrode2UsageElozo:=GVL.nElectrode2Usage;
				GVL.nElectrode2UsageWarnElozo:=GVL.nElectrode2UsageWarn;
				GVL.nElectrode2UsageMaxElozo:=GVL.nElectrode2UsageMax;
				GVL.nElectrode3UsageElozo:=GVL.nElectrode3Usage;
				GVL.nElectrode3UsageWarnElozo:=GVL.nElectrode3UsageWarn;
				GVL.nElectrode3UsageMaxElozo:=GVL.nElectrode3UsageMax;
				GVL.nHegFejTisztCiklusokElozo:=GVL.nHegFejTisztCiklusok;
				GVL.nHegFejTisztProgramElozo:=GVL.nHegFejTisztProgram;
				// A hegesztési paraméterek figyelmeztető ill. riasztó színeinek beállítása, ha szükséges:
				IF GVL.nElectrode1Usage>GVL.nElectrode1UsageMax THEN
					GVL.nElectrode1AlarmColor:=16#FFFF0000; // piros
				ELSE
					GVL.nElectrode1AlarmColor:=16#FFFFFF00; //sárga
				END_IF
				IF GVL.nElectrode2Usage>GVL.nElectrode2UsageMax THEN
					GVL.nElectrode2AlarmColor:=16#FFFF0000;
				ELSE
					GVL.nElectrode2AlarmColor:=16#FFFFFF00;
				END_IF
				IF GVL.nElectrode3Usage>GVL.nElectrode3UsageMax THEN
					GVL.nElectrode3AlarmColor:=16#FFFF0000;
				ELSE
					GVL.nElectrode3AlarmColor:=16#FFFFFF00;
				END_IF
				iStateS:=12;
			END_IF
		ELSE
			iStateS:=103;
		END_IF
	13:	// Settings fájl zárásának kezdeményezése
		bSettingsCloseExecute:=TRUE;
		iStateS:=14;
	14:	// Várakozás a busy jelre
		IF bSettingsCloseBusy=TRUE THEN
			iStateS:=15;
		END_IF
	15:	// Várakozás a fájlzárás befejeztére
		IF bSettingsCloseBusy=FALSE THEN
			bSettingsCloseExecute:=FALSE;
			iStateS:=16;
		END_IF
	16:	// Fájlzárás sikerességének vizsgálata
		IF bSettingsCloseError=FALSE THEN
			bSettingsReadReady:=TRUE;	
			iStateS:=2;
		ELSE
			iStateS:=104;
		END_IF

END_CASE


PartsOpen(
		sNetId:='',
		sPathName:='C:\637\Init\Parts.ini',
		nMode:=nPartsOpenMode,
		ePath:=PATH_GENERIC,
		bExecute:=bPartsOpenExecute,
		tTimeout:=T#5S,
		bBusy=>bPartsOpenBusy,
		bError=>bPartsOpenError,
		nErrId=>nPartsOpenError,
		hFile=>hPartsFile
		);
		
PartsPutStr(
		sNetId:='',
		hFile:=hPartsFile,
		sLine:=sPartsString,
		bExecute:=bPartsPutStrExecute,
		tTimeout:=T#1S,
		bBusy=>bPartsPutStrBusy,
		bError=>bPartsPutStrError,
		nErrId=>nPartsPutStrError);
		
PartsGetStr(
		sNetId:='',
		hFile:=hPartsFile,
		bExecute:=bPartsGetStrExecute,
		tTimeout:=T#1S,
		bBusy=>bPartsGetStrBusy,
		bError=>bPartsGetStrError,
		nErrId=>nPartsGetStrError,
		sLine=>sPartsGetStr,
		bEOF=>bGetStrPartsEOF
);
		
PartsClose(
		sNetId:='',
		hFile:=hPartsFile,
		bExecute:=bPartsCloseExecute,
		tTimeout:=T#5S,
		bBusy=>bPartsCloseBusy,
		bError=>bPartsCloseError,
		nErrId=>nPartsCloseError
		);

SettingsOpen(
		sNetId:='',
		sPathName:='C:\637\Init\Settings.ini',
		nMode:=nSettingsOpenMode,
		ePath:=PATH_GENERIC,
		bExecute:=bSettingsOpenExecute,
		tTimeout:=T#5S,
		bBusy=>bSettingsOpenBusy,
		bError=>bSettingsOpenError,
		nErrId=>nSettingsOpenError,
		hFile=>hSettingsFile
		);
		
SettingsPutStr(
		sNetId:='',
		hFile:=hSettingsFile,
		sLine:=sSettingsString,
		bExecute:=bSettingsPutStrExecute,
		tTimeout:=T#1S,
		bBusy=>bSettingsPutStrBusy,
		bError=>bSettingsPutStrError,
		nErrId=>nSettingsPutStrError);
		
